(* IEC 61131-3 sources: TIA2AX/tests/V18/test_projects/expected/HW_2200330/ST10_PLC, 7 files *)

(* ---- HwIdentifiers.st ---- *)
TYPE
	HwIdentifiers : WORD
	(
		ST10_PLC_Rail_0 :=	WORD#256,
		ST10_PLC :=	WORD#48,
		ST10_PLC_Card_reader_writer_1 :=	WORD#51,
		ST10_PLC_CPU_display_1 :=	WORD#54,
		ST10_PLC_OPC_UA_1 :=	WORD#117,
		ST10_PLC_DP_interface_1 :=	WORD#60,
		ST10_PLC_PROFINET_interface_1 :=	WORD#64,
		ST10_PLC_PROFINET_interface_1_Port_1 :=	WORD#65,
		ST10_PLC_PROFINET_interface_1_Port_2 :=	WORD#66,
		ST10_PLC_PROFINET_interface_2 :=	WORD#72,
		ST10_PLC_PROFINET_interface_2_Port_1 :=	WORD#73,
		ST10_Switch_SCALANCE_X_rack :=	WORD#479,
		ST10_Switch :=	WORD#480,
		ST10_Switch_ST10_Switch :=	WORD#481,
		ST10_Switch_SCALANCE_interface_1 :=	WORD#482,
		ST10_Switch_SCALANCE_interface_1_Port_1 :=	WORD#483,
		ST10_Switch_SCALANCE_interface_1_Port_2 :=	WORD#484,
		ST10_Switch_SCALANCE_interface_1_Port_3 :=	WORD#485,
		ST10_Switch_SCALANCE_interface_1_Port_4 :=	WORD#486,
		ST10_Switch_SCALANCE_interface_1_Port_5 :=	WORD#487,
		ST10_Switch_SCALANCE_interface_1_Port_6 :=	WORD#488,
		ST10_Switch_SCALANCE_interface_1_Port_7 :=	WORD#489,
		ST10_Switch_SCALANCE_interface_1_Port_8 :=	WORD#490,
		ST10_Switch_SCALANCE_interface_1_Port_9 :=	WORD#491,
		ST10_Switch_SCALANCE_interface_1_Port_10 :=	WORD#492,
		ST10_Switch_SCALANCE_interface_1_Port_11 :=	WORD#493,
		ST10_Switch_SCALANCE_interface_1_Port_12 :=	WORD#494,
		ST10_Switch_SCALANCE_interface_1_Port_13 :=	WORD#495,
		ST10_Switch_SCALANCE_interface_1_Port_14 :=	WORD#496,
		ST10_Switch_SCALANCE_interface_1_Port_15 :=	WORD#497,
		ST10_Switch_SCALANCE_interface_1_Port_16 :=	WORD#498,
		ST10_ET200SP_Rack_0 :=	WORD#395,
		ST10_ET200SP :=	WORD#396,
		ST10_ET200SP_ST10_ET200SP :=	WORD#397,
		ST10_ET200SP_PROFINET_interface :=	WORD#259,
		ST10_ET200SP_PROFINET_interface_Port_1 :=	WORD#260,
		ST10_ET200SP_PROFINET_interface_Port_2 :=	WORD#261,
		ST10_ET200SP_BA_2xRJ45 :=	WORD#260,
		ST10_ET200SP_CM_AS_i_Master_ST_1 :=	WORD#274,
		ST10_ET200SP_DI_8x24VDC_ST_1 :=	WORD#264,
		ST10_ET200SP_DI_16x24VDC_ST_2 :=	WORD#265,
		ST10_ET200SP_DI_16x24VDC_ST_3 :=	WORD#266,
		ST10_ET200SP_DI_8x24VDC_ST_2 :=	WORD#267,
		ST10_ET200SP_DQ_8x24VDC_0_5A_ST_1 :=	WORD#268,
		ST10_ET200SP_DQ_8x24VDC_0_5A_ST_2 :=	WORD#269,
		ST10_ET200SP_DQ_8x24VDC_0_5A_ST_3 :=	WORD#270,
		ST10_ET200SP_DQ_8x24VDC_0_5A_ST_4 :=	WORD#271,
		ST10_ET200SP_CM_4xIO_Link_1 :=	WORD#272,
		ST10_ET200SP_Servermodul_1 :=	WORD#273,
		ST10_ET200SP_2_Rack_0 :=	WORD#399,
		ST10_ET200SP_2 :=	WORD#400,
		ST10_ET200SP_2_ST10_ET200SP_2 :=	WORD#401,
		ST10_ET200SP_2_PROFINET_interface :=	WORD#402,
		ST10_ET200SP_2_PROFINET_interface_Port_1 :=	WORD#404,
		ST10_ET200SP_2_PROFINET_interface_Port_2 :=	WORD#403,
		ST10_ET200SP_2_BA_2xRJ45 :=	WORD#404,
		ST10_ET200SP_2_21FM1 :=	WORD#405,
		ST10_ET200SP_2_21FM2 :=	WORD#406,
		ST10_ET200SP_2_21FM3 :=	WORD#407,
		ST10_ET200SP_2_21FM4 :=	WORD#408,
		ST10_ET200SP_2_21FM5 :=	WORD#409,
		ST10_ET200SP_2_21FM6 :=	WORD#410,
		ST10_ET200SP_2_21FM7 :=	WORD#411,
		ST10_ET200SP_2_21FM8 :=	WORD#412,
		ST10_ET200SP_2_21FM9 :=	WORD#413,
		ST10_ET200SP_2_21FM10 :=	WORD#414,
		ST10_ET200SP_2_21FM11 :=	WORD#415,
		ST10_ET200SP_2_21FM12 :=	WORD#416,
		ST10_ET200SP_2_22FM1 :=	WORD#417,
		ST10_ET200SP_2_22FM2 :=	WORD#418,
		ST10_ET200SP_2_22FM3 :=	WORD#419,
		ST10_ET200SP_2_22FM4 :=	WORD#420,
		ST10_ET200SP_2_22FM5 :=	WORD#421,
		ST10_ET200SP_2_22FM6 :=	WORD#422,
		ST10_ET200SP_2_22FM7 :=	WORD#423,
		ST10_ET200SP_2_22FM8 :=	WORD#424,
		ST10_ET200SP_2_22FM9 :=	WORD#425,
		ST10_ET200SP_2_22FM10 :=	WORD#426,
		ST10_ET200SP_2_22FM11 :=	WORD#427,
		ST10_ET200SP_2_22FM12 :=	WORD#428,
		ST10_ET200SP_2_22FM13 :=	WORD#429,
		ST10_ET200SP_2_Servermodul :=	WORD#430,
		ST10_CPX_PN_IO_Interface :=	WORD#434,
		ST10_CPX_PN_IO_Interface_Port_1 :=	WORD#435,
		ST10_CPX_PN_IO_Interface_Port_2 :=	WORD#436,
		ST10_CPX_CPX :=	WORD#437,
		ST10_CPX_MPA1S_VMPA1_FB_EMS_8_8DO_1 :=	WORD#438,
		ST10_CPX_MPA2G_VMPA2_FB_EMG_4_4DO_1 :=	WORD#439,
		ST10_1_DM260_Rack :=	WORD#441,
		ST10_1_DM260 :=	WORD#442,
		ST10_1_DM260_Interface :=	WORD#443,
		ST10_1_DM260_Interface_Port_1 :=	WORD#444,
		ST10_1_DM260_DataMan_260 :=	WORD#445,
		ST10_1_DM260_Acquisition_Control_1 :=	WORD#446,
		ST10_1_DM260_Acquisition_Status_1 :=	WORD#447,
		ST10_1_DM260_Results_Control_1 :=	WORD#448,
		ST10_1_DM260_Results_Status_1 :=	WORD#449,
		ST10_1_DM260_Soft_Event_Control_1 :=	WORD#450,
		ST10_1_DM260_User_Data_64_bytes_1 :=	WORD#451,
		ST10_1_DM260_Result_Data_64_bytes_1 :=	WORD#452,
		ST10_1_DM260_Turned_Rack :=	WORD#454,
		ST10_1_DM260_Turned :=	WORD#455,
		ST10_1_DM260_Turned_Interface :=	WORD#456,
		ST10_1_DM260_Turned_Interface_Port_1 :=	WORD#457,
		ST10_1_DM260_Turned_DataMan_260 :=	WORD#458,
		ST10_1_DM260_Turned_Acquisition_Control_1 :=	WORD#459,
		ST10_1_DM260_Turned_Acquisition_Status_1 :=	WORD#460,
		ST10_1_DM260_Turned_Results_Control_1 :=	WORD#461,
		ST10_1_DM260_Turned_Results_Status_1 :=	WORD#462,
		ST10_1_DM260_Turned_Soft_Event_Control_1 :=	WORD#463,
		ST10_1_DM260_Turned_User_Data_64_bytes_1 :=	WORD#464,
		ST10_1_DM260_Turned_Result_Data_64_bytes_1 :=	WORD#465,
		NONE:= WORD#0
	);
END_TYPE

(* ---- HwInputs.st ---- *)
TYPE
	HwInputs : STRUCT
		ST10_ET200SP_CM_AS_i_Master_ST_1 AT %B300 : ARRAY[0..63] OF BYTE;
		ST10_ET200SP_DI_8x24VDC_ST_1 AT %B0 : BYTE;
		ST10_ET200SP_DI_16x24VDC_ST_2 AT %B1 : WORD;
		ST10_ET200SP_DI_16x24VDC_ST_3 AT %B3 : WORD;
		ST10_ET200SP_DI_8x24VDC_ST_2 AT %B5 : BYTE;
		ST10_ET200SP_CM_4xIO_Link_1 AT %B100 : ARRAY[0..31] OF BYTE;
		ST10_ET200SP_2_21FM1 AT %B600 : DWORD;
		ST10_ET200SP_2_21FM2 AT %B604 : DWORD;
		ST10_ET200SP_2_21FM3 AT %B652 : DWORD;
		ST10_ET200SP_2_21FM4 AT %B612 : DWORD;
		ST10_ET200SP_2_21FM5 AT %B616 : DWORD;
		ST10_ET200SP_2_21FM6 AT %B620 : DWORD;
		ST10_ET200SP_2_21FM7 AT %B624 : DWORD;
		ST10_ET200SP_2_21FM8 AT %B628 : DWORD;
		ST10_ET200SP_2_21FM9 AT %B632 : DWORD;
		ST10_ET200SP_2_21FM10 AT %B636 : DWORD;
		ST10_ET200SP_2_21FM11 AT %B640 : DWORD;
		ST10_ET200SP_2_21FM12 AT %B644 : DWORD;
		ST10_ET200SP_2_22FM1 AT %B648 : DWORD;
		ST10_ET200SP_2_22FM2 AT %B608 : DWORD;
		ST10_ET200SP_2_22FM3 AT %B696 : DWORD;
		ST10_ET200SP_2_22FM4 AT %B660 : DWORD;
		ST10_ET200SP_2_22FM5 AT %B664 : DWORD;
		ST10_ET200SP_2_22FM6 AT %B668 : DWORD;
		ST10_ET200SP_2_22FM7 AT %B672 : DWORD;
		ST10_ET200SP_2_22FM8 AT %B676 : DWORD;
		ST10_ET200SP_2_22FM9 AT %B656 : DWORD;
		ST10_ET200SP_2_22FM10 AT %B684 : DWORD;
		ST10_ET200SP_2_22FM11 AT %B688 : DWORD;
		ST10_ET200SP_2_22FM12 AT %B692 : DWORD;
		ST10_ET200SP_2_22FM13 AT %B680 : DWORD;
		ST10_1_DM260_Acquisition_Status_1 AT %B1000 : ARRAY[0..2] OF BYTE;
		ST10_1_DM260_Results_Status_1 AT %B1003 : BYTE;
		ST10_1_DM260_Soft_Event_Control_1 AT %B1004 : BYTE;
		ST10_1_DM260_Result_Data_64_bytes_1 AT %B1010 : ARRAY[0..71] OF BYTE;
		ST10_1_DM260_Turned_Acquisition_Status_1 AT %B1200 : ARRAY[0..2] OF BYTE;
		ST10_1_DM260_Turned_Results_Status_1 AT %B1203 : BYTE;
		ST10_1_DM260_Turned_Soft_Event_Control_1 AT %B1204 : BYTE;
		ST10_1_DM260_Turned_Result_Data_64_bytes_1 AT %B1210 : ARRAY[0..71] OF BYTE;
	END_STRUCT;
END_TYPE

(* ---- HwOutputs.st ---- *)
TYPE
	HwOutputs : STRUCT
		ST10_ET200SP_CM_AS_i_Master_ST_1 AT %B300 : ARRAY[0..63] OF BYTE;
		ST10_ET200SP_DQ_8x24VDC_0_5A_ST_1 AT %B0 : BYTE;
		ST10_ET200SP_DQ_8x24VDC_0_5A_ST_2 AT %B1 : BYTE;
		ST10_ET200SP_DQ_8x24VDC_0_5A_ST_3 AT %B2 : BYTE;
		ST10_ET200SP_DQ_8x24VDC_0_5A_ST_4 AT %B3 : BYTE;
		ST10_ET200SP_CM_4xIO_Link_1 AT %B100 : ARRAY[0..31] OF BYTE;
		ST10_ET200SP_2_21FM1 AT %B600 : WORD;
		ST10_ET200SP_2_21FM2 AT %B604 : WORD;
		ST10_ET200SP_2_21FM3 AT %B652 : WORD;
		ST10_ET200SP_2_21FM4 AT %B612 : WORD;
		ST10_ET200SP_2_21FM5 AT %B616 : WORD;
		ST10_ET200SP_2_21FM6 AT %B620 : WORD;
		ST10_ET200SP_2_21FM7 AT %B624 : WORD;
		ST10_ET200SP_2_21FM8 AT %B628 : WORD;
		ST10_ET200SP_2_21FM9 AT %B632 : WORD;
		ST10_ET200SP_2_21FM10 AT %B636 : WORD;
		ST10_ET200SP_2_21FM11 AT %B640 : WORD;
		ST10_ET200SP_2_21FM12 AT %B644 : WORD;
		ST10_ET200SP_2_22FM1 AT %B648 : WORD;
		ST10_ET200SP_2_22FM2 AT %B608 : WORD;
		ST10_ET200SP_2_22FM3 AT %B692 : WORD;
		ST10_ET200SP_2_22FM4 AT %B660 : WORD;
		ST10_ET200SP_2_22FM5 AT %B664 : WORD;
		ST10_ET200SP_2_22FM6 AT %B668 : WORD;
		ST10_ET200SP_2_22FM7 AT %B672 : WORD;
		ST10_ET200SP_2_22FM8 AT %B676 : WORD;
		ST10_ET200SP_2_22FM9 AT %B656 : WORD;
		ST10_ET200SP_2_22FM10 AT %B684 : WORD;
		ST10_ET200SP_2_22FM11 AT %B688 : WORD;
		ST10_ET200SP_2_22FM12 AT %B690 : WORD;
		ST10_ET200SP_2_22FM13 AT %B680 : WORD;
		ST10_CPX_MPA1S_VMPA1_FB_EMS_8_8DO_1 AT %B200 : BYTE;
		ST10_CPX_MPA2G_VMPA2_FB_EMG_4_4DO_1 AT %B201 : BYTE;
		ST10_1_DM260_Acquisition_Control_1 AT %B1000 : BYTE;
		ST10_1_DM260_Results_Control_1 AT %B1001 : BYTE;
		ST10_1_DM260_Soft_Event_Control_1 AT %B1002 : BYTE;
		ST10_1_DM260_User_Data_64_bytes_1 AT %B1010 : ARRAY[0..67] OF BYTE;
		ST10_1_DM260_Turned_Acquisition_Control_1 AT %B1200 : BYTE;
		ST10_1_DM260_Turned_Results_Control_1 AT %B1203 : BYTE;
		ST10_1_DM260_Turned_Soft_Event_Control_1 AT %B1204 : BYTE;
		ST10_1_DM260_Turned_User_Data_64_bytes_1 AT %B1210 : ARRAY[0..67] OF BYTE;
	END_STRUCT;
END_TYPE

(* ---- PlcInputs.st ---- *)
TYPE
	PlcInputs : STRUCT
		ST10_ET200SP_CM_AS_i_Master_ST_1 : ARRAY[0..63] OF BYTE;
		ST10_ET200SP_DI_8x24VDC_ST_1 : BYTE;
		ST10_ET200SP_DI_16x24VDC_ST_2 : WORD;
		ST10_ET200SP_DI_16x24VDC_ST_3 : WORD;
		ST10_ET200SP_DI_8x24VDC_ST_2 : BYTE;
		ST10_ET200SP_CM_4xIO_Link_1 : ARRAY[0..31] OF BYTE;
		ST10_ET200SP_2_21FM1 : DWORD;
		ST10_ET200SP_2_21FM2 : DWORD;
		ST10_ET200SP_2_21FM3 : DWORD;
		ST10_ET200SP_2_21FM4 : DWORD;
		ST10_ET200SP_2_21FM5 : DWORD;
		ST10_ET200SP_2_21FM6 : DWORD;
		ST10_ET200SP_2_21FM7 : DWORD;
		ST10_ET200SP_2_21FM8 : DWORD;
		ST10_ET200SP_2_21FM9 : DWORD;
		ST10_ET200SP_2_21FM10 : DWORD;
		ST10_ET200SP_2_21FM11 : DWORD;
		ST10_ET200SP_2_21FM12 : DWORD;
		ST10_ET200SP_2_22FM1 : DWORD;
		ST10_ET200SP_2_22FM2 : DWORD;
		ST10_ET200SP_2_22FM3 : DWORD;
		ST10_ET200SP_2_22FM4 : DWORD;
		ST10_ET200SP_2_22FM5 : DWORD;
		ST10_ET200SP_2_22FM6 : DWORD;
		ST10_ET200SP_2_22FM7 : DWORD;
		ST10_ET200SP_2_22FM8 : DWORD;
		ST10_ET200SP_2_22FM9 : DWORD;
		ST10_ET200SP_2_22FM10 : DWORD;
		ST10_ET200SP_2_22FM11 : DWORD;
		ST10_ET200SP_2_22FM12 : DWORD;
		ST10_ET200SP_2_22FM13 : DWORD;
		ST10_1_DM260_Acquisition_Status_1 : ARRAY[0..2] OF BYTE;
		ST10_1_DM260_Results_Status_1 : BYTE;
		ST10_1_DM260_Soft_Event_Control_1 : BYTE;
		ST10_1_DM260_Result_Data_64_bytes_1 : ARRAY[0..71] OF BYTE;
		ST10_1_DM260_Turned_Acquisition_Status_1 : ARRAY[0..2] OF BYTE;
		ST10_1_DM260_Turned_Results_Status_1 : BYTE;
		ST10_1_DM260_Turned_Soft_Event_Control_1 : BYTE;
		ST10_1_DM260_Turned_Result_Data_64_bytes_1 : ARRAY[0..71] OF BYTE;
	END_STRUCT;
END_TYPE

(* ---- PlcOutputs.st ---- *)
TYPE
	PlcOutputs : STRUCT
		ST10_ET200SP_CM_AS_i_Master_ST_1 : ARRAY[0..63] OF BYTE;
		ST10_ET200SP_DQ_8x24VDC_0_5A_ST_1 : BYTE;
		ST10_ET200SP_DQ_8x24VDC_0_5A_ST_2 : BYTE;
		ST10_ET200SP_DQ_8x24VDC_0_5A_ST_3 : BYTE;
		ST10_ET200SP_DQ_8x24VDC_0_5A_ST_4 : BYTE;
		ST10_ET200SP_CM_4xIO_Link_1 : ARRAY[0..31] OF BYTE;
		ST10_ET200SP_2_21FM1 : WORD;
		ST10_ET200SP_2_21FM2 : WORD;
		ST10_ET200SP_2_21FM3 : WORD;
		ST10_ET200SP_2_21FM4 : WORD;
		ST10_ET200SP_2_21FM5 : WORD;
		ST10_ET200SP_2_21FM6 : WORD;
		ST10_ET200SP_2_21FM7 : WORD;
		ST10_ET200SP_2_21FM8 : WORD;
		ST10_ET200SP_2_21FM9 : WORD;
		ST10_ET200SP_2_21FM10 : WORD;
		ST10_ET200SP_2_21FM11 : WORD;
		ST10_ET200SP_2_21FM12 : WORD;
		ST10_ET200SP_2_22FM1 : WORD;
		ST10_ET200SP_2_22FM2 : WORD;
		ST10_ET200SP_2_22FM3 : WORD;
		ST10_ET200SP_2_22FM4 : WORD;
		ST10_ET200SP_2_22FM5 : WORD;
		ST10_ET200SP_2_22FM6 : WORD;
		ST10_ET200SP_2_22FM7 : WORD;
		ST10_ET200SP_2_22FM8 : WORD;
		ST10_ET200SP_2_22FM9 : WORD;
		ST10_ET200SP_2_22FM10 : WORD;
		ST10_ET200SP_2_22FM11 : WORD;
		ST10_ET200SP_2_22FM12 : WORD;
		ST10_ET200SP_2_22FM13 : WORD;
		ST10_CPX_MPA1S_VMPA1_FB_EMS_8_8DO_1 : BYTE;
		ST10_CPX_MPA2G_VMPA2_FB_EMG_4_4DO_1 : BYTE;
		ST10_1_DM260_Acquisition_Control_1 : BYTE;
		ST10_1_DM260_Results_Control_1 : BYTE;
		ST10_1_DM260_Soft_Event_Control_1 : BYTE;
		ST10_1_DM260_User_Data_64_bytes_1 : ARRAY[0..67] OF BYTE;
		ST10_1_DM260_Turned_Acquisition_Control_1 : BYTE;
		ST10_1_DM260_Turned_Results_Control_1 : BYTE;
		ST10_1_DM260_Turned_Soft_Event_Control_1 : BYTE;
		ST10_1_DM260_Turned_User_Data_64_bytes_1 : ARRAY[0..67] OF BYTE;
	END_STRUCT;
END_TYPE

(* ---- CopyInputs.st ---- *)
FUNCTION CopyInputs
	VAR_EXTERNAL
		HwInputs : HwInputs;
		PlcInputs : PlcInputs;
	END_VAR
	PlcInputs.ST10_ET200SP_CM_AS_i_Master_ST_1[0] := HwInputs.ST10_ET200SP_CM_AS_i_Master_ST_1[0];
	PlcInputs.ST10_ET200SP_CM_AS_i_Master_ST_1[1] := HwInputs.ST10_ET200SP_CM_AS_i_Master_ST_1[1];
	PlcInputs.ST10_ET200SP_CM_AS_i_Master_ST_1[2] := HwInputs.ST10_ET200SP_CM_AS_i_Master_ST_1[2];
	PlcInputs.ST10_ET200SP_CM_AS_i_Master_ST_1[3] := HwInputs.ST10_ET200SP_CM_AS_i_Master_ST_1[3];
	PlcInputs.ST10_ET200SP_CM_AS_i_Master_ST_1[4] := HwInputs.ST10_ET200SP_CM_AS_i_Master_ST_1[4];
	PlcInputs.ST10_ET200SP_CM_AS_i_Master_ST_1[5] := HwInputs.ST10_ET200SP_CM_AS_i_Master_ST_1[5];
	PlcInputs.ST10_ET200SP_CM_AS_i_Master_ST_1[6] := HwInputs.ST10_ET200SP_CM_AS_i_Master_ST_1[6];
	PlcInputs.ST10_ET200SP_CM_AS_i_Master_ST_1[7] := HwInputs.ST10_ET200SP_CM_AS_i_Master_ST_1[7];
	PlcInputs.ST10_ET200SP_CM_AS_i_Master_ST_1[8] := HwInputs.ST10_ET200SP_CM_AS_i_Master_ST_1[8];
	PlcInputs.ST10_ET200SP_CM_AS_i_Master_ST_1[9] := HwInputs.ST10_ET200SP_CM_AS_i_Master_ST_1[9];
	PlcInputs.ST10_ET200SP_CM_AS_i_Master_ST_1[10] := HwInputs.ST10_ET200SP_CM_AS_i_Master_ST_1[10];
	PlcInputs.ST10_ET200SP_CM_AS_i_Master_ST_1[11] := HwInputs.ST10_ET200SP_CM_AS_i_Master_ST_1[11];
	PlcInputs.ST10_ET200SP_CM_AS_i_Master_ST_1[12] := HwInputs.ST10_ET200SP_CM_AS_i_Master_ST_1[12];
	PlcInputs.ST10_ET200SP_CM_AS_i_Master_ST_1[13] := HwInputs.ST10_ET200SP_CM_AS_i_Master_ST_1[13];
	PlcInputs.ST10_ET200SP_CM_AS_i_Master_ST_1[14] := HwInputs.ST10_ET200SP_CM_AS_i_Master_ST_1[14];
	PlcInputs.ST10_ET200SP_CM_AS_i_Master_ST_1[15] := HwInputs.ST10_ET200SP_CM_AS_i_Master_ST_1[15];
	PlcInputs.ST10_ET200SP_CM_AS_i_Master_ST_1[16] := HwInputs.ST10_ET200SP_CM_AS_i_Master_ST_1[16];
	PlcInputs.ST10_ET200SP_CM_AS_i_Master_ST_1[17] := HwInputs.ST10_ET200SP_CM_AS_i_Master_ST_1[17];
	PlcInputs.ST10_ET200SP_CM_AS_i_Master_ST_1[18] := HwInputs.ST10_ET200SP_CM_AS_i_Master_ST_1[18];
	PlcInputs.ST10_ET200SP_CM_AS_i_Master_ST_1[19] := HwInputs.ST10_ET200SP_CM_AS_i_Master_ST_1[19];
	PlcInputs.ST10_ET200SP_CM_AS_i_Master_ST_1[20] := HwInputs.ST10_ET200SP_CM_AS_i_Master_ST_1[20];
	PlcInputs.ST10_ET200SP_CM_AS_i_Master_ST_1[21] := HwInputs.ST10_ET200SP_CM_AS_i_Master_ST_1[21];
	PlcInputs.ST10_ET200SP_CM_AS_i_Master_ST_1[22] := HwInputs.ST10_ET200SP_CM_AS_i_Master_ST_1[22];
	PlcInputs.ST10_ET200SP_CM_AS_i_Master_ST_1[23] := HwInputs.ST10_ET200SP_CM_AS_i_Master_ST_1[23];
	PlcInputs.ST10_ET200SP_CM_AS_i_Master_ST_1[24] := HwInputs.ST10_ET200SP_CM_AS_i_Master_ST_1[24];
	PlcInputs.ST10_ET200SP_CM_AS_i_Master_ST_1[25] := HwInputs.ST10_ET200SP_CM_AS_i_Master_ST_1[25];
	PlcInputs.ST10_ET200SP_CM_AS_i_Master_ST_1[26] := HwInputs.ST10_ET200SP_CM_AS_i_Master_ST_1[26];
	PlcInputs.ST10_ET200SP_CM_AS_i_Master_ST_1[27] := HwInputs.ST10_ET200SP_CM_AS_i_Master_ST_1[27];
	PlcInputs.ST10_ET200SP_CM_AS_i_Master_ST_1[28] := HwInputs.ST10_ET200SP_CM_AS_i_Master_ST_1[28];
	PlcInputs.ST10_ET200SP_CM_AS_i_Master_ST_1[29] := HwInputs.ST10_ET200SP_CM_AS_i_Master_ST_1[29];
	PlcInputs.ST10_ET200SP_CM_AS_i_Master_ST_1[30] := HwInputs.ST10_ET200SP_CM_AS_i_Master_ST_1[30];
	PlcInputs.ST10_ET200SP_CM_AS_i_Master_ST_1[31] := HwInputs.ST10_ET200SP_CM_AS_i_Master_ST_1[31];
	PlcInputs.ST10_ET200SP_CM_AS_i_Master_ST_1[32] := HwInputs.ST10_ET200SP_CM_AS_i_Master_ST_1[32];
	PlcInputs.ST10_ET200SP_CM_AS_i_Master_ST_1[33] := HwInputs.ST10_ET200SP_CM_AS_i_Master_ST_1[33];
	PlcInputs.ST10_ET200SP_CM_AS_i_Master_ST_1[34] := HwInputs.ST10_ET200SP_CM_AS_i_Master_ST_1[34];
	PlcInputs.ST10_ET200SP_CM_AS_i_Master_ST_1[35] := HwInputs.ST10_ET200SP_CM_AS_i_Master_ST_1[35];
	PlcInputs.ST10_ET200SP_CM_AS_i_Master_ST_1[36] := HwInputs.ST10_ET200SP_CM_AS_i_Master_ST_1[36];
	PlcInputs.ST10_ET200SP_CM_AS_i_Master_ST_1[37] := HwInputs.ST10_ET200SP_CM_AS_i_Master_ST_1[37];
	PlcInputs.ST10_ET200SP_CM_AS_i_Master_ST_1[38] := HwInputs.ST10_ET200SP_CM_AS_i_Master_ST_1[38];
	PlcInputs.ST10_ET200SP_CM_AS_i_Master_ST_1[39] := HwInputs.ST10_ET200SP_CM_AS_i_Master_ST_1[39];
	PlcInputs.ST10_ET200SP_CM_AS_i_Master_ST_1[40] := HwInputs.ST10_ET200SP_CM_AS_i_Master_ST_1[40];
	PlcInputs.ST10_ET200SP_CM_AS_i_Master_ST_1[41] := HwInputs.ST10_ET200SP_CM_AS_i_Master_ST_1[41];
	PlcInputs.ST10_ET200SP_CM_AS_i_Master_ST_1[42] := HwInputs.ST10_ET200SP_CM_AS_i_Master_ST_1[42];
	PlcInputs.ST10_ET200SP_CM_AS_i_Master_ST_1[43] := HwInputs.ST10_ET200SP_CM_AS_i_Master_ST_1[43];
	PlcInputs.ST10_ET200SP_CM_AS_i_Master_ST_1[44] := HwInputs.ST10_ET200SP_CM_AS_i_Master_ST_1[44];
	PlcInputs.ST10_ET200SP_CM_AS_i_Master_ST_1[45] := HwInputs.ST10_ET200SP_CM_AS_i_Master_ST_1[45];
	PlcInputs.ST10_ET200SP_CM_AS_i_Master_ST_1[46] := HwInputs.ST10_ET200SP_CM_AS_i_Master_ST_1[46];
	PlcInputs.ST10_ET200SP_CM_AS_i_Master_ST_1[47] := HwInputs.ST10_ET200SP_CM_AS_i_Master_ST_1[47];
	PlcInputs.ST10_ET200SP_CM_AS_i_Master_ST_1[48] := HwInputs.ST10_ET200SP_CM_AS_i_Master_ST_1[48];
	PlcInputs.ST10_ET200SP_CM_AS_i_Master_ST_1[49] := HwInputs.ST10_ET200SP_CM_AS_i_Master_ST_1[49];
	PlcInputs.ST10_ET200SP_CM_AS_i_Master_ST_1[50] := HwInputs.ST10_ET200SP_CM_AS_i_Master_ST_1[50];
	PlcInputs.ST10_ET200SP_CM_AS_i_Master_ST_1[51] := HwInputs.ST10_ET200SP_CM_AS_i_Master_ST_1[51];
	PlcInputs.ST10_ET200SP_CM_AS_i_Master_ST_1[52] := HwInputs.ST10_ET200SP_CM_AS_i_Master_ST_1[52];
	PlcInputs.ST10_ET200SP_CM_AS_i_Master_ST_1[53] := HwInputs.ST10_ET200SP_CM_AS_i_Master_ST_1[53];
	PlcInputs.ST10_ET200SP_CM_AS_i_Master_ST_1[54] := HwInputs.ST10_ET200SP_CM_AS_i_Master_ST_1[54];
	PlcInputs.ST10_ET200SP_CM_AS_i_Master_ST_1[55] := HwInputs.ST10_ET200SP_CM_AS_i_Master_ST_1[55];
	PlcInputs.ST10_ET200SP_CM_AS_i_Master_ST_1[56] := HwInputs.ST10_ET200SP_CM_AS_i_Master_ST_1[56];
	PlcInputs.ST10_ET200SP_CM_AS_i_Master_ST_1[57] := HwInputs.ST10_ET200SP_CM_AS_i_Master_ST_1[57];
	PlcInputs.ST10_ET200SP_CM_AS_i_Master_ST_1[58] := HwInputs.ST10_ET200SP_CM_AS_i_Master_ST_1[58];
	PlcInputs.ST10_ET200SP_CM_AS_i_Master_ST_1[59] := HwInputs.ST10_ET200SP_CM_AS_i_Master_ST_1[59];
	PlcInputs.ST10_ET200SP_CM_AS_i_Master_ST_1[60] := HwInputs.ST10_ET200SP_CM_AS_i_Master_ST_1[60];
	PlcInputs.ST10_ET200SP_CM_AS_i_Master_ST_1[61] := HwInputs.ST10_ET200SP_CM_AS_i_Master_ST_1[61];
	PlcInputs.ST10_ET200SP_CM_AS_i_Master_ST_1[62] := HwInputs.ST10_ET200SP_CM_AS_i_Master_ST_1[62];
	PlcInputs.ST10_ET200SP_CM_AS_i_Master_ST_1[63] := HwInputs.ST10_ET200SP_CM_AS_i_Master_ST_1[63];
	PlcInputs.ST10_ET200SP_DI_8x24VDC_ST_1 := HwInputs.ST10_ET200SP_DI_8x24VDC_ST_1;
	PlcInputs.ST10_ET200SP_DI_16x24VDC_ST_2 := HwInputs.ST10_ET200SP_DI_16x24VDC_ST_2;
	PlcInputs.ST10_ET200SP_DI_16x24VDC_ST_3 := HwInputs.ST10_ET200SP_DI_16x24VDC_ST_3;
	PlcInputs.ST10_ET200SP_DI_8x24VDC_ST_2 := HwInputs.ST10_ET200SP_DI_8x24VDC_ST_2;
	PlcInputs.ST10_ET200SP_CM_4xIO_Link_1[0] := HwInputs.ST10_ET200SP_CM_4xIO_Link_1[0];
	PlcInputs.ST10_ET200SP_CM_4xIO_Link_1[1] := HwInputs.ST10_ET200SP_CM_4xIO_Link_1[1];
	PlcInputs.ST10_ET200SP_CM_4xIO_Link_1[2] := HwInputs.ST10_ET200SP_CM_4xIO_Link_1[2];
	PlcInputs.ST10_ET200SP_CM_4xIO_Link_1[3] := HwInputs.ST10_ET200SP_CM_4xIO_Link_1[3];
	PlcInputs.ST10_ET200SP_CM_4xIO_Link_1[4] := HwInputs.ST10_ET200SP_CM_4xIO_Link_1[4];
	PlcInputs.ST10_ET200SP_CM_4xIO_Link_1[5] := HwInputs.ST10_ET200SP_CM_4xIO_Link_1[5];
	PlcInputs.ST10_ET200SP_CM_4xIO_Link_1[6] := HwInputs.ST10_ET200SP_CM_4xIO_Link_1[6];
	PlcInputs.ST10_ET200SP_CM_4xIO_Link_1[7] := HwInputs.ST10_ET200SP_CM_4xIO_Link_1[7];
	PlcInputs.ST10_ET200SP_CM_4xIO_Link_1[8] := HwInputs.ST10_ET200SP_CM_4xIO_Link_1[8];
	PlcInputs.ST10_ET200SP_CM_4xIO_Link_1[9] := HwInputs.ST10_ET200SP_CM_4xIO_Link_1[9];
	PlcInputs.ST10_ET200SP_CM_4xIO_Link_1[10] := HwInputs.ST10_ET200SP_CM_4xIO_Link_1[10];
	PlcInputs.ST10_ET200SP_CM_4xIO_Link_1[11] := HwInputs.ST10_ET200SP_CM_4xIO_Link_1[11];
	PlcInputs.ST10_ET200SP_CM_4xIO_Link_1[12] := HwInputs.ST10_ET200SP_CM_4xIO_Link_1[12];
	PlcInputs.ST10_ET200SP_CM_4xIO_Link_1[13] := HwInputs.ST10_ET200SP_CM_4xIO_Link_1[13];
	PlcInputs.ST10_ET200SP_CM_4xIO_Link_1[14] := HwInputs.ST10_ET200SP_CM_4xIO_Link_1[14];
	PlcInputs.ST10_ET200SP_CM_4xIO_Link_1[15] := HwInputs.ST10_ET200SP_CM_4xIO_Link_1[15];
	PlcInputs.ST10_ET200SP_CM_4xIO_Link_1[16] := HwInputs.ST10_ET200SP_CM_4xIO_Link_1[16];
	PlcInputs.ST10_ET200SP_CM_4xIO_Link_1[17] := HwInputs.ST10_ET200SP_CM_4xIO_Link_1[17];
	PlcInputs.ST10_ET200SP_CM_4xIO_Link_1[18] := HwInputs.ST10_ET200SP_CM_4xIO_Link_1[18];
	PlcInputs.ST10_ET200SP_CM_4xIO_Link_1[19] := HwInputs.ST10_ET200SP_CM_4xIO_Link_1[19];
	PlcInputs.ST10_ET200SP_CM_4xIO_Link_1[20] := HwInputs.ST10_ET200SP_CM_4xIO_Link_1[20];
	PlcInputs.ST10_ET200SP_CM_4xIO_Link_1[21] := HwInputs.ST10_ET200SP_CM_4xIO_Link_1[21];
	PlcInputs.ST10_ET200SP_CM_4xIO_Link_1[22] := HwInputs.ST10_ET200SP_CM_4xIO_Link_1[22];
	PlcInputs.ST10_ET200SP_CM_4xIO_Link_1[23] := HwInputs.ST10_ET200SP_CM_4xIO_Link_1[23];
	PlcInputs.ST10_ET200SP_CM_4xIO_Link_1[24] := HwInputs.ST10_ET200SP_CM_4xIO_Link_1[24];
	PlcInputs.ST10_ET200SP_CM_4xIO_Link_1[25] := HwInputs.ST10_ET200SP_CM_4xIO_Link_1[25];
	PlcInputs.ST10_ET200SP_CM_4xIO_Link_1[26] := HwInputs.ST10_ET200SP_CM_4xIO_Link_1[26];
	PlcInputs.ST10_ET200SP_CM_4xIO_Link_1[27] := HwInputs.ST10_ET200SP_CM_4xIO_Link_1[27];
	PlcInputs.ST10_ET200SP_CM_4xIO_Link_1[28] := HwInputs.ST10_ET200SP_CM_4xIO_Link_1[28];
	PlcInputs.ST10_ET200SP_CM_4xIO_Link_1[29] := HwInputs.ST10_ET200SP_CM_4xIO_Link_1[29];
	PlcInputs.ST10_ET200SP_CM_4xIO_Link_1[30] := HwInputs.ST10_ET200SP_CM_4xIO_Link_1[30];
	PlcInputs.ST10_ET200SP_CM_4xIO_Link_1[31] := HwInputs.ST10_ET200SP_CM_4xIO_Link_1[31];
	PlcInputs.ST10_ET200SP_2_21FM1 := HwInputs.ST10_ET200SP_2_21FM1;
	PlcInputs.ST10_ET200SP_2_21FM2 := HwInputs.ST10_ET200SP_2_21FM2;
	PlcInputs.ST10_ET200SP_2_21FM3 := HwInputs.ST10_ET200SP_2_21FM3;
	PlcInputs.ST10_ET200SP_2_21FM4 := HwInputs.ST10_ET200SP_2_21FM4;
	PlcInputs.ST10_ET200SP_2_21FM5 := HwInputs.ST10_ET200SP_2_21FM5;
	PlcInputs.ST10_ET200SP_2_21FM6 := HwInputs.ST10_ET200SP_2_21FM6;
	PlcInputs.ST10_ET200SP_2_21FM7 := HwInputs.ST10_ET200SP_2_21FM7;
	PlcInputs.ST10_ET200SP_2_21FM8 := HwInputs.ST10_ET200SP_2_21FM8;
	PlcInputs.ST10_ET200SP_2_21FM9 := HwInputs.ST10_ET200SP_2_21FM9;
	PlcInputs.ST10_ET200SP_2_21FM10 := HwInputs.ST10_ET200SP_2_21FM10;
	PlcInputs.ST10_ET200SP_2_21FM11 := HwInputs.ST10_ET200SP_2_21FM11;
	PlcInputs.ST10_ET200SP_2_21FM12 := HwInputs.ST10_ET200SP_2_21FM12;
	PlcInputs.ST10_ET200SP_2_22FM1 := HwInputs.ST10_ET200SP_2_22FM1;
	PlcInputs.ST10_ET200SP_2_22FM2 := HwInputs.ST10_ET200SP_2_22FM2;
	PlcInputs.ST10_ET200SP_2_22FM3 := HwInputs.ST10_ET200SP_2_22FM3;
	PlcInputs.ST10_ET200SP_2_22FM4 := HwInputs.ST10_ET200SP_2_22FM4;
	PlcInputs.ST10_ET200SP_2_22FM5 := HwInputs.ST10_ET200SP_2_22FM5;
	PlcInputs.ST10_ET200SP_2_22FM6 := HwInputs.ST10_ET200SP_2_22FM6;
	PlcInputs.ST10_ET200SP_2_22FM7 := HwInputs.ST10_ET200SP_2_22FM7;
	PlcInputs.ST10_ET200SP_2_22FM8 := HwInputs.ST10_ET200SP_2_22FM8;
	PlcInputs.ST10_ET200SP_2_22FM9 := HwInputs.ST10_ET200SP_2_22FM9;
	PlcInputs.ST10_ET200SP_2_22FM10 := HwInputs.ST10_ET200SP_2_22FM10;
	PlcInputs.ST10_ET200SP_2_22FM11 := HwInputs.ST10_ET200SP_2_22FM11;
	PlcInputs.ST10_ET200SP_2_22FM12 := HwInputs.ST10_ET200SP_2_22FM12;
	PlcInputs.ST10_ET200SP_2_22FM13 := HwInputs.ST10_ET200SP_2_22FM13;
	PlcInputs.ST10_1_DM260_Acquisition_Status_1[0] := HwInputs.ST10_1_DM260_Acquisition_Status_1[0];
	PlcInputs.ST10_1_DM260_Acquisition_Status_1[1] := HwInputs.ST10_1_DM260_Acquisition_Status_1[1];
	PlcInputs.ST10_1_DM260_Acquisition_Status_1[2] := HwInputs.ST10_1_DM260_Acquisition_Status_1[2];
	PlcInputs.ST10_1_DM260_Results_Status_1 := HwInputs.ST10_1_DM260_Results_Status_1;
	PlcInputs.ST10_1_DM260_Soft_Event_Control_1 := HwInputs.ST10_1_DM260_Soft_Event_Control_1;
	PlcInputs.ST10_1_DM260_Result_Data_64_bytes_1[0] := HwInputs.ST10_1_DM260_Result_Data_64_bytes_1[0];
	PlcInputs.ST10_1_DM260_Result_Data_64_bytes_1[1] := HwInputs.ST10_1_DM260_Result_Data_64_bytes_1[1];
	PlcInputs.ST10_1_DM260_Result_Data_64_bytes_1[2] := HwInputs.ST10_1_DM260_Result_Data_64_bytes_1[2];
	PlcInputs.ST10_1_DM260_Result_Data_64_bytes_1[3] := HwInputs.ST10_1_DM260_Result_Data_64_bytes_1[3];
	PlcInputs.ST10_1_DM260_Result_Data_64_bytes_1[4] := HwInputs.ST10_1_DM260_Result_Data_64_bytes_1[4];
	PlcInputs.ST10_1_DM260_Result_Data_64_bytes_1[5] := HwInputs.ST10_1_DM260_Result_Data_64_bytes_1[5];
	PlcInputs.ST10_1_DM260_Result_Data_64_bytes_1[6] := HwInputs.ST10_1_DM260_Result_Data_64_bytes_1[6];
	PlcInputs.ST10_1_DM260_Result_Data_64_bytes_1[7] := HwInputs.ST10_1_DM260_Result_Data_64_bytes_1[7];
	PlcInputs.ST10_1_DM260_Result_Data_64_bytes_1[8] := HwInputs.ST10_1_DM260_Result_Data_64_bytes_1[8];
	PlcInputs.ST10_1_DM260_Result_Data_64_bytes_1[9] := HwInputs.ST10_1_DM260_Result_Data_64_bytes_1[9];
	PlcInputs.ST10_1_DM260_Result_Data_64_bytes_1[10] := HwInputs.ST10_1_DM260_Result_Data_64_bytes_1[10];
	PlcInputs.ST10_1_DM260_Result_Data_64_bytes_1[11] := HwInputs.ST10_1_DM260_Result_Data_64_bytes_1[11];
	PlcInputs.ST10_1_DM260_Result_Data_64_bytes_1[12] := HwInputs.ST10_1_DM260_Result_Data_64_bytes_1[12];
	PlcInputs.ST10_1_DM260_Result_Data_64_bytes_1[13] := HwInputs.ST10_1_DM260_Result_Data_64_bytes_1[13];
	PlcInputs.ST10_1_DM260_Result_Data_64_bytes_1[14] := HwInputs.ST10_1_DM260_Result_Data_64_bytes_1[14];
	PlcInputs.ST10_1_DM260_Result_Data_64_bytes_1[15] := HwInputs.ST10_1_DM260_Result_Data_64_bytes_1[15];
	PlcInputs.ST10_1_DM260_Result_Data_64_bytes_1[16] := HwInputs.ST10_1_DM260_Result_Data_64_bytes_1[16];
	PlcInputs.ST10_1_DM260_Result_Data_64_bytes_1[17] := HwInputs.ST10_1_DM260_Result_Data_64_bytes_1[17];
	PlcInputs.ST10_1_DM260_Result_Data_64_bytes_1[18] := HwInputs.ST10_1_DM260_Result_Data_64_bytes_1[18];
	PlcInputs.ST10_1_DM260_Result_Data_64_bytes_1[19] := HwInputs.ST10_1_DM260_Result_Data_64_bytes_1[19];
	PlcInputs.ST10_1_DM260_Result_Data_64_bytes_1[20] := HwInputs.ST10_1_DM260_Result_Data_64_bytes_1[20];
	PlcInputs.ST10_1_DM260_Result_Data_64_bytes_1[21] := HwInputs.ST10_1_DM260_Result_Data_64_bytes_1[21];
	PlcInputs.ST10_1_DM260_Result_Data_64_bytes_1[22] := HwInputs.ST10_1_DM260_Result_Data_64_bytes_1[22];
	PlcInputs.ST10_1_DM260_Result_Data_64_bytes_1[23] := HwInputs.ST10_1_DM260_Result_Data_64_bytes_1[23];
	PlcInputs.ST10_1_DM260_Result_Data_64_bytes_1[24] := HwInputs.ST10_1_DM260_Result_Data_64_bytes_1[24];
	PlcInputs.ST10_1_DM260_Result_Data_64_bytes_1[25] := HwInputs.ST10_1_DM260_Result_Data_64_bytes_1[25];
	PlcInputs.ST10_1_DM260_Result_Data_64_bytes_1[26] := HwInputs.ST10_1_DM260_Result_Data_64_bytes_1[26];
	PlcInputs.ST10_1_DM260_Result_Data_64_bytes_1[27] := HwInputs.ST10_1_DM260_Result_Data_64_bytes_1[27];
	PlcInputs.ST10_1_DM260_Result_Data_64_bytes_1[28] := HwInputs.ST10_1_DM260_Result_Data_64_bytes_1[28];
	PlcInputs.ST10_1_DM260_Result_Data_64_bytes_1[29] := HwInputs.ST10_1_DM260_Result_Data_64_bytes_1[29];
	PlcInputs.ST10_1_DM260_Result_Data_64_bytes_1[30] := HwInputs.ST10_1_DM260_Result_Data_64_bytes_1[30];
	PlcInputs.ST10_1_DM260_Result_Data_64_bytes_1[31] := HwInputs.ST10_1_DM260_Result_Data_64_bytes_1[31];
	PlcInputs.ST10_1_DM260_Result_Data_64_bytes_1[32] := HwInputs.ST10_1_DM260_Result_Data_64_bytes_1[32];
	PlcInputs.ST10_1_DM260_Result_Data_64_bytes_1[33] := HwInputs.ST10_1_DM260_Result_Data_64_bytes_1[33];
	PlcInputs.ST10_1_DM260_Result_Data_64_bytes_1[34] := HwInputs.ST10_1_DM260_Result_Data_64_bytes_1[34];
	PlcInputs.ST10_1_DM260_Result_Data_64_bytes_1[35] := HwInputs.ST10_1_DM260_Result_Data_64_bytes_1[35];
	PlcInputs.ST10_1_DM260_Result_Data_64_bytes_1[36] := HwInputs.ST10_1_DM260_Result_Data_64_bytes_1[36];
	PlcInputs.ST10_1_DM260_Result_Data_64_bytes_1[37] := HwInputs.ST10_1_DM260_Result_Data_64_bytes_1[37];
	PlcInputs.ST10_1_DM260_Result_Data_64_bytes_1[38] := HwInputs.ST10_1_DM260_Result_Data_64_bytes_1[38];
	PlcInputs.ST10_1_DM260_Result_Data_64_bytes_1[39] := HwInputs.ST10_1_DM260_Result_Data_64_bytes_1[39];
	PlcInputs.ST10_1_DM260_Result_Data_64_bytes_1[40] := HwInputs.ST10_1_DM260_Result_Data_64_bytes_1[40];
	PlcInputs.ST10_1_DM260_Result_Data_64_bytes_1[41] := HwInputs.ST10_1_DM260_Result_Data_64_bytes_1[41];
	PlcInputs.ST10_1_DM260_Result_Data_64_bytes_1[42] := HwInputs.ST10_1_DM260_Result_Data_64_bytes_1[42];
	PlcInputs.ST10_1_DM260_Result_Data_64_bytes_1[43] := HwInputs.ST10_1_DM260_Result_Data_64_bytes_1[43];
	PlcInputs.ST10_1_DM260_Result_Data_64_bytes_1[44] := HwInputs.ST10_1_DM260_Result_Data_64_bytes_1[44];
	PlcInputs.ST10_1_DM260_Result_Data_64_bytes_1[45] := HwInputs.ST10_1_DM260_Result_Data_64_bytes_1[45];
	PlcInputs.ST10_1_DM260_Result_Data_64_bytes_1[46] := HwInputs.ST10_1_DM260_Result_Data_64_bytes_1[46];
	PlcInputs.ST10_1_DM260_Result_Data_64_bytes_1[47] := HwInputs.ST10_1_DM260_Result_Data_64_bytes_1[47];
	PlcInputs.ST10_1_DM260_Result_Data_64_bytes_1[48] := HwInputs.ST10_1_DM260_Result_Data_64_bytes_1[48];
	PlcInputs.ST10_1_DM260_Result_Data_64_bytes_1[49] := HwInputs.ST10_1_DM260_Result_Data_64_bytes_1[49];
	PlcInputs.ST10_1_DM260_Result_Data_64_bytes_1[50] := HwInputs.ST10_1_DM260_Result_Data_64_bytes_1[50];
	PlcInputs.ST10_1_DM260_Result_Data_64_bytes_1[51] := HwInputs.ST10_1_DM260_Result_Data_64_bytes_1[51];
	PlcInputs.ST10_1_DM260_Result_Data_64_bytes_1[52] := HwInputs.ST10_1_DM260_Result_Data_64_bytes_1[52];
	PlcInputs.ST10_1_DM260_Result_Data_64_bytes_1[53] := HwInputs.ST10_1_DM260_Result_Data_64_bytes_1[53];
	PlcInputs.ST10_1_DM260_Result_Data_64_bytes_1[54] := HwInputs.ST10_1_DM260_Result_Data_64_bytes_1[54];
	PlcInputs.ST10_1_DM260_Result_Data_64_bytes_1[55] := HwInputs.ST10_1_DM260_Result_Data_64_bytes_1[55];
	PlcInputs.ST10_1_DM260_Result_Data_64_bytes_1[56] := HwInputs.ST10_1_DM260_Result_Data_64_bytes_1[56];
	PlcInputs.ST10_1_DM260_Result_Data_64_bytes_1[57] := HwInputs.ST10_1_DM260_Result_Data_64_bytes_1[57];
	PlcInputs.ST10_1_DM260_Result_Data_64_bytes_1[58] := HwInputs.ST10_1_DM260_Result_Data_64_bytes_1[58];
	PlcInputs.ST10_1_DM260_Result_Data_64_bytes_1[59] := HwInputs.ST10_1_DM260_Result_Data_64_bytes_1[59];
	PlcInputs.ST10_1_DM260_Result_Data_64_bytes_1[60] := HwInputs.ST10_1_DM260_Result_Data_64_bytes_1[60];
	PlcInputs.ST10_1_DM260_Result_Data_64_bytes_1[61] := HwInputs.ST10_1_DM260_Result_Data_64_bytes_1[61];
	PlcInputs.ST10_1_DM260_Result_Data_64_bytes_1[62] := HwInputs.ST10_1_DM260_Result_Data_64_bytes_1[62];
	PlcInputs.ST10_1_DM260_Result_Data_64_bytes_1[63] := HwInputs.ST10_1_DM260_Result_Data_64_bytes_1[63];
	PlcInputs.ST10_1_DM260_Result_Data_64_bytes_1[64] := HwInputs.ST10_1_DM260_Result_Data_64_bytes_1[64];
	PlcInputs.ST10_1_DM260_Result_Data_64_bytes_1[65] := HwInputs.ST10_1_DM260_Result_Data_64_bytes_1[65];
	PlcInputs.ST10_1_DM260_Result_Data_64_bytes_1[66] := HwInputs.ST10_1_DM260_Result_Data_64_bytes_1[66];
	PlcInputs.ST10_1_DM260_Result_Data_64_bytes_1[67] := HwInputs.ST10_1_DM260_Result_Data_64_bytes_1[67];
	PlcInputs.ST10_1_DM260_Result_Data_64_bytes_1[68] := HwInputs.ST10_1_DM260_Result_Data_64_bytes_1[68];
	PlcInputs.ST10_1_DM260_Result_Data_64_bytes_1[69] := HwInputs.ST10_1_DM260_Result_Data_64_bytes_1[69];
	PlcInputs.ST10_1_DM260_Result_Data_64_bytes_1[70] := HwInputs.ST10_1_DM260_Result_Data_64_bytes_1[70];
	PlcInputs.ST10_1_DM260_Result_Data_64_bytes_1[71] := HwInputs.ST10_1_DM260_Result_Data_64_bytes_1[71];
	PlcInputs.ST10_1_DM260_Turned_Acquisition_Status_1[0] := HwInputs.ST10_1_DM260_Turned_Acquisition_Status_1[0];
	PlcInputs.ST10_1_DM260_Turned_Acquisition_Status_1[1] := HwInputs.ST10_1_DM260_Turned_Acquisition_Status_1[1];
	PlcInputs.ST10_1_DM260_Turned_Acquisition_Status_1[2] := HwInputs.ST10_1_DM260_Turned_Acquisition_Status_1[2];
	PlcInputs.ST10_1_DM260_Turned_Results_Status_1 := HwInputs.ST10_1_DM260_Turned_Results_Status_1;
	PlcInputs.ST10_1_DM260_Turned_Soft_Event_Control_1 := HwInputs.ST10_1_DM260_Turned_Soft_Event_Control_1;
	PlcInputs.ST10_1_DM260_Turned_Result_Data_64_bytes_1[0] := HwInputs.ST10_1_DM260_Turned_Result_Data_64_bytes_1[0];
	PlcInputs.ST10_1_DM260_Turned_Result_Data_64_bytes_1[1] := HwInputs.ST10_1_DM260_Turned_Result_Data_64_bytes_1[1];
	PlcInputs.ST10_1_DM260_Turned_Result_Data_64_bytes_1[2] := HwInputs.ST10_1_DM260_Turned_Result_Data_64_bytes_1[2];
	PlcInputs.ST10_1_DM260_Turned_Result_Data_64_bytes_1[3] := HwInputs.ST10_1_DM260_Turned_Result_Data_64_bytes_1[3];
	PlcInputs.ST10_1_DM260_Turned_Result_Data_64_bytes_1[4] := HwInputs.ST10_1_DM260_Turned_Result_Data_64_bytes_1[4];
	PlcInputs.ST10_1_DM260_Turned_Result_Data_64_bytes_1[5] := HwInputs.ST10_1_DM260_Turned_Result_Data_64_bytes_1[5];
	PlcInputs.ST10_1_DM260_Turned_Result_Data_64_bytes_1[6] := HwInputs.ST10_1_DM260_Turned_Result_Data_64_bytes_1[6];
	PlcInputs.ST10_1_DM260_Turned_Result_Data_64_bytes_1[7] := HwInputs.ST10_1_DM260_Turned_Result_Data_64_bytes_1[7];
	PlcInputs.ST10_1_DM260_Turned_Result_Data_64_bytes_1[8] := HwInputs.ST10_1_DM260_Turned_Result_Data_64_bytes_1[8];
	PlcInputs.ST10_1_DM260_Turned_Result_Data_64_bytes_1[9] := HwInputs.ST10_1_DM260_Turned_Result_Data_64_bytes_1[9];
	PlcInputs.ST10_1_DM260_Turned_Result_Data_64_bytes_1[10] := HwInputs.ST10_1_DM260_Turned_Result_Data_64_bytes_1[10];
	PlcInputs.ST10_1_DM260_Turned_Result_Data_64_bytes_1[11] := HwInputs.ST10_1_DM260_Turned_Result_Data_64_bytes_1[11];
	PlcInputs.ST10_1_DM260_Turned_Result_Data_64_bytes_1[12] := HwInputs.ST10_1_DM260_Turned_Result_Data_64_bytes_1[12];
	PlcInputs.ST10_1_DM260_Turned_Result_Data_64_bytes_1[13] := HwInputs.ST10_1_DM260_Turned_Result_Data_64_bytes_1[13];
	PlcInputs.ST10_1_DM260_Turned_Result_Data_64_bytes_1[14] := HwInputs.ST10_1_DM260_Turned_Result_Data_64_bytes_1[14];
	PlcInputs.ST10_1_DM260_Turned_Result_Data_64_bytes_1[15] := HwInputs.ST10_1_DM260_Turned_Result_Data_64_bytes_1[15];
	PlcInputs.ST10_1_DM260_Turned_Result_Data_64_bytes_1[16] := HwInputs.ST10_1_DM260_Turned_Result_Data_64_bytes_1[16];
	PlcInputs.ST10_1_DM260_Turned_Result_Data_64_bytes_1[17] := HwInputs.ST10_1_DM260_Turned_Result_Data_64_bytes_1[17];
	PlcInputs.ST10_1_DM260_Turned_Result_Data_64_bytes_1[18] := HwInputs.ST10_1_DM260_Turned_Result_Data_64_bytes_1[18];
	PlcInputs.ST10_1_DM260_Turned_Result_Data_64_bytes_1[19] := HwInputs.ST10_1_DM260_Turned_Result_Data_64_bytes_1[19];
	PlcInputs.ST10_1_DM260_Turned_Result_Data_64_bytes_1[20] := HwInputs.ST10_1_DM260_Turned_Result_Data_64_bytes_1[20];
	PlcInputs.ST10_1_DM260_Turned_Result_Data_64_bytes_1[21] := HwInputs.ST10_1_DM260_Turned_Result_Data_64_bytes_1[21];
	PlcInputs.ST10_1_DM260_Turned_Result_Data_64_bytes_1[22] := HwInputs.ST10_1_DM260_Turned_Result_Data_64_bytes_1[22];
	PlcInputs.ST10_1_DM260_Turned_Result_Data_64_bytes_1[23] := HwInputs.ST10_1_DM260_Turned_Result_Data_64_bytes_1[23];
	PlcInputs.ST10_1_DM260_Turned_Result_Data_64_bytes_1[24] := HwInputs.ST10_1_DM260_Turned_Result_Data_64_bytes_1[24];
	PlcInputs.ST10_1_DM260_Turned_Result_Data_64_bytes_1[25] := HwInputs.ST10_1_DM260_Turned_Result_Data_64_bytes_1[25];
	PlcInputs.ST10_1_DM260_Turned_Result_Data_64_bytes_1[26] := HwInputs.ST10_1_DM260_Turned_Result_Data_64_bytes_1[26];
	PlcInputs.ST10_1_DM260_Turned_Result_Data_64_bytes_1[27] := HwInputs.ST10_1_DM260_Turned_Result_Data_64_bytes_1[27];
	PlcInputs.ST10_1_DM260_Turned_Result_Data_64_bytes_1[28] := HwInputs.ST10_1_DM260_Turned_Result_Data_64_bytes_1[28];
	PlcInputs.ST10_1_DM260_Turned_Result_Data_64_bytes_1[29] := HwInputs.ST10_1_DM260_Turned_Result_Data_64_bytes_1[29];
	PlcInputs.ST10_1_DM260_Turned_Result_Data_64_bytes_1[30] := HwInputs.ST10_1_DM260_Turned_Result_Data_64_bytes_1[30];
	PlcInputs.ST10_1_DM260_Turned_Result_Data_64_bytes_1[31] := HwInputs.ST10_1_DM260_Turned_Result_Data_64_bytes_1[31];
	PlcInputs.ST10_1_DM260_Turned_Result_Data_64_bytes_1[32] := HwInputs.ST10_1_DM260_Turned_Result_Data_64_bytes_1[32];
	PlcInputs.ST10_1_DM260_Turned_Result_Data_64_bytes_1[33] := HwInputs.ST10_1_DM260_Turned_Result_Data_64_bytes_1[33];
	PlcInputs.ST10_1_DM260_Turned_Result_Data_64_bytes_1[34] := HwInputs.ST10_1_DM260_Turned_Result_Data_64_bytes_1[34];
	PlcInputs.ST10_1_DM260_Turned_Result_Data_64_bytes_1[35] := HwInputs.ST10_1_DM260_Turned_Result_Data_64_bytes_1[35];
	PlcInputs.ST10_1_DM260_Turned_Result_Data_64_bytes_1[36] := HwInputs.ST10_1_DM260_Turned_Result_Data_64_bytes_1[36];
	PlcInputs.ST10_1_DM260_Turned_Result_Data_64_bytes_1[37] := HwInputs.ST10_1_DM260_Turned_Result_Data_64_bytes_1[37];
	PlcInputs.ST10_1_DM260_Turned_Result_Data_64_bytes_1[38] := HwInputs.ST10_1_DM260_Turned_Result_Data_64_bytes_1[38];
	PlcInputs.ST10_1_DM260_Turned_Result_Data_64_bytes_1[39] := HwInputs.ST10_1_DM260_Turned_Result_Data_64_bytes_1[39];
	PlcInputs.ST10_1_DM260_Turned_Result_Data_64_bytes_1[40] := HwInputs.ST10_1_DM260_Turned_Result_Data_64_bytes_1[40];
	PlcInputs.ST10_1_DM260_Turned_Result_Data_64_bytes_1[41] := HwInputs.ST10_1_DM260_Turned_Result_Data_64_bytes_1[41];
	PlcInputs.ST10_1_DM260_Turned_Result_Data_64_bytes_1[42] := HwInputs.ST10_1_DM260_Turned_Result_Data_64_bytes_1[42];
	PlcInputs.ST10_1_DM260_Turned_Result_Data_64_bytes_1[43] := HwInputs.ST10_1_DM260_Turned_Result_Data_64_bytes_1[43];
	PlcInputs.ST10_1_DM260_Turned_Result_Data_64_bytes_1[44] := HwInputs.ST10_1_DM260_Turned_Result_Data_64_bytes_1[44];
	PlcInputs.ST10_1_DM260_Turned_Result_Data_64_bytes_1[45] := HwInputs.ST10_1_DM260_Turned_Result_Data_64_bytes_1[45];
	PlcInputs.ST10_1_DM260_Turned_Result_Data_64_bytes_1[46] := HwInputs.ST10_1_DM260_Turned_Result_Data_64_bytes_1[46];
	PlcInputs.ST10_1_DM260_Turned_Result_Data_64_bytes_1[47] := HwInputs.ST10_1_DM260_Turned_Result_Data_64_bytes_1[47];
	PlcInputs.ST10_1_DM260_Turned_Result_Data_64_bytes_1[48] := HwInputs.ST10_1_DM260_Turned_Result_Data_64_bytes_1[48];
	PlcInputs.ST10_1_DM260_Turned_Result_Data_64_bytes_1[49] := HwInputs.ST10_1_DM260_Turned_Result_Data_64_bytes_1[49];
	PlcInputs.ST10_1_DM260_Turned_Result_Data_64_bytes_1[50] := HwInputs.ST10_1_DM260_Turned_Result_Data_64_bytes_1[50];
	PlcInputs.ST10_1_DM260_Turned_Result_Data_64_bytes_1[51] := HwInputs.ST10_1_DM260_Turned_Result_Data_64_bytes_1[51];
	PlcInputs.ST10_1_DM260_Turned_Result_Data_64_bytes_1[52] := HwInputs.ST10_1_DM260_Turned_Result_Data_64_bytes_1[52];
	PlcInputs.ST10_1_DM260_Turned_Result_Data_64_bytes_1[53] := HwInputs.ST10_1_DM260_Turned_Result_Data_64_bytes_1[53];
	PlcInputs.ST10_1_DM260_Turned_Result_Data_64_bytes_1[54] := HwInputs.ST10_1_DM260_Turned_Result_Data_64_bytes_1[54];
	PlcInputs.ST10_1_DM260_Turned_Result_Data_64_bytes_1[55] := HwInputs.ST10_1_DM260_Turned_Result_Data_64_bytes_1[55];
	PlcInputs.ST10_1_DM260_Turned_Result_Data_64_bytes_1[56] := HwInputs.ST10_1_DM260_Turned_Result_Data_64_bytes_1[56];
	PlcInputs.ST10_1_DM260_Turned_Result_Data_64_bytes_1[57] := HwInputs.ST10_1_DM260_Turned_Result_Data_64_bytes_1[57];
	PlcInputs.ST10_1_DM260_Turned_Result_Data_64_bytes_1[58] := HwInputs.ST10_1_DM260_Turned_Result_Data_64_bytes_1[58];
	PlcInputs.ST10_1_DM260_Turned_Result_Data_64_bytes_1[59] := HwInputs.ST10_1_DM260_Turned_Result_Data_64_bytes_1[59];
	PlcInputs.ST10_1_DM260_Turned_Result_Data_64_bytes_1[60] := HwInputs.ST10_1_DM260_Turned_Result_Data_64_bytes_1[60];
	PlcInputs.ST10_1_DM260_Turned_Result_Data_64_bytes_1[61] := HwInputs.ST10_1_DM260_Turned_Result_Data_64_bytes_1[61];
	PlcInputs.ST10_1_DM260_Turned_Result_Data_64_bytes_1[62] := HwInputs.ST10_1_DM260_Turned_Result_Data_64_bytes_1[62];
	PlcInputs.ST10_1_DM260_Turned_Result_Data_64_bytes_1[63] := HwInputs.ST10_1_DM260_Turned_Result_Data_64_bytes_1[63];
	PlcInputs.ST10_1_DM260_Turned_Result_Data_64_bytes_1[64] := HwInputs.ST10_1_DM260_Turned_Result_Data_64_bytes_1[64];
	PlcInputs.ST10_1_DM260_Turned_Result_Data_64_bytes_1[65] := HwInputs.ST10_1_DM260_Turned_Result_Data_64_bytes_1[65];
	PlcInputs.ST10_1_DM260_Turned_Result_Data_64_bytes_1[66] := HwInputs.ST10_1_DM260_Turned_Result_Data_64_bytes_1[66];
	PlcInputs.ST10_1_DM260_Turned_Result_Data_64_bytes_1[67] := HwInputs.ST10_1_DM260_Turned_Result_Data_64_bytes_1[67];
	PlcInputs.ST10_1_DM260_Turned_Result_Data_64_bytes_1[68] := HwInputs.ST10_1_DM260_Turned_Result_Data_64_bytes_1[68];
	PlcInputs.ST10_1_DM260_Turned_Result_Data_64_bytes_1[69] := HwInputs.ST10_1_DM260_Turned_Result_Data_64_bytes_1[69];
	PlcInputs.ST10_1_DM260_Turned_Result_Data_64_bytes_1[70] := HwInputs.ST10_1_DM260_Turned_Result_Data_64_bytes_1[70];
	PlcInputs.ST10_1_DM260_Turned_Result_Data_64_bytes_1[71] := HwInputs.ST10_1_DM260_Turned_Result_Data_64_bytes_1[71];
END_FUNCTION

(* ---- CopyOutputs.st ---- *)
FUNCTION CopyOutputs
	VAR_EXTERNAL
		HwOutputs : HwOutputs;
		PlcOutputs : PlcOutputs;
	END_VAR
	HwOutputs.ST10_ET200SP_CM_AS_i_Master_ST_1[0] := PlcOutputs.ST10_ET200SP_CM_AS_i_Master_ST_1[0];
	HwOutputs.ST10_ET200SP_CM_AS_i_Master_ST_1[1] := PlcOutputs.ST10_ET200SP_CM_AS_i_Master_ST_1[1];
	HwOutputs.ST10_ET200SP_CM_AS_i_Master_ST_1[2] := PlcOutputs.ST10_ET200SP_CM_AS_i_Master_ST_1[2];
	HwOutputs.ST10_ET200SP_CM_AS_i_Master_ST_1[3] := PlcOutputs.ST10_ET200SP_CM_AS_i_Master_ST_1[3];
	HwOutputs.ST10_ET200SP_CM_AS_i_Master_ST_1[4] := PlcOutputs.ST10_ET200SP_CM_AS_i_Master_ST_1[4];
	HwOutputs.ST10_ET200SP_CM_AS_i_Master_ST_1[5] := PlcOutputs.ST10_ET200SP_CM_AS_i_Master_ST_1[5];
	HwOutputs.ST10_ET200SP_CM_AS_i_Master_ST_1[6] := PlcOutputs.ST10_ET200SP_CM_AS_i_Master_ST_1[6];
	HwOutputs.ST10_ET200SP_CM_AS_i_Master_ST_1[7] := PlcOutputs.ST10_ET200SP_CM_AS_i_Master_ST_1[7];
	HwOutputs.ST10_ET200SP_CM_AS_i_Master_ST_1[8] := PlcOutputs.ST10_ET200SP_CM_AS_i_Master_ST_1[8];
	HwOutputs.ST10_ET200SP_CM_AS_i_Master_ST_1[9] := PlcOutputs.ST10_ET200SP_CM_AS_i_Master_ST_1[9];
	HwOutputs.ST10_ET200SP_CM_AS_i_Master_ST_1[10] := PlcOutputs.ST10_ET200SP_CM_AS_i_Master_ST_1[10];
	HwOutputs.ST10_ET200SP_CM_AS_i_Master_ST_1[11] := PlcOutputs.ST10_ET200SP_CM_AS_i_Master_ST_1[11];
	HwOutputs.ST10_ET200SP_CM_AS_i_Master_ST_1[12] := PlcOutputs.ST10_ET200SP_CM_AS_i_Master_ST_1[12];
	HwOutputs.ST10_ET200SP_CM_AS_i_Master_ST_1[13] := PlcOutputs.ST10_ET200SP_CM_AS_i_Master_ST_1[13];
	HwOutputs.ST10_ET200SP_CM_AS_i_Master_ST_1[14] := PlcOutputs.ST10_ET200SP_CM_AS_i_Master_ST_1[14];
	HwOutputs.ST10_ET200SP_CM_AS_i_Master_ST_1[15] := PlcOutputs.ST10_ET200SP_CM_AS_i_Master_ST_1[15];
	HwOutputs.ST10_ET200SP_CM_AS_i_Master_ST_1[16] := PlcOutputs.ST10_ET200SP_CM_AS_i_Master_ST_1[16];
	HwOutputs.ST10_ET200SP_CM_AS_i_Master_ST_1[17] := PlcOutputs.ST10_ET200SP_CM_AS_i_Master_ST_1[17];
	HwOutputs.ST10_ET200SP_CM_AS_i_Master_ST_1[18] := PlcOutputs.ST10_ET200SP_CM_AS_i_Master_ST_1[18];
	HwOutputs.ST10_ET200SP_CM_AS_i_Master_ST_1[19] := PlcOutputs.ST10_ET200SP_CM_AS_i_Master_ST_1[19];
	HwOutputs.ST10_ET200SP_CM_AS_i_Master_ST_1[20] := PlcOutputs.ST10_ET200SP_CM_AS_i_Master_ST_1[20];
	HwOutputs.ST10_ET200SP_CM_AS_i_Master_ST_1[21] := PlcOutputs.ST10_ET200SP_CM_AS_i_Master_ST_1[21];
	HwOutputs.ST10_ET200SP_CM_AS_i_Master_ST_1[22] := PlcOutputs.ST10_ET200SP_CM_AS_i_Master_ST_1[22];
	HwOutputs.ST10_ET200SP_CM_AS_i_Master_ST_1[23] := PlcOutputs.ST10_ET200SP_CM_AS_i_Master_ST_1[23];
	HwOutputs.ST10_ET200SP_CM_AS_i_Master_ST_1[24] := PlcOutputs.ST10_ET200SP_CM_AS_i_Master_ST_1[24];
	HwOutputs.ST10_ET200SP_CM_AS_i_Master_ST_1[25] := PlcOutputs.ST10_ET200SP_CM_AS_i_Master_ST_1[25];
	HwOutputs.ST10_ET200SP_CM_AS_i_Master_ST_1[26] := PlcOutputs.ST10_ET200SP_CM_AS_i_Master_ST_1[26];
	HwOutputs.ST10_ET200SP_CM_AS_i_Master_ST_1[27] := PlcOutputs.ST10_ET200SP_CM_AS_i_Master_ST_1[27];
	HwOutputs.ST10_ET200SP_CM_AS_i_Master_ST_1[28] := PlcOutputs.ST10_ET200SP_CM_AS_i_Master_ST_1[28];
	HwOutputs.ST10_ET200SP_CM_AS_i_Master_ST_1[29] := PlcOutputs.ST10_ET200SP_CM_AS_i_Master_ST_1[29];
	HwOutputs.ST10_ET200SP_CM_AS_i_Master_ST_1[30] := PlcOutputs.ST10_ET200SP_CM_AS_i_Master_ST_1[30];
	HwOutputs.ST10_ET200SP_CM_AS_i_Master_ST_1[31] := PlcOutputs.ST10_ET200SP_CM_AS_i_Master_ST_1[31];
	HwOutputs.ST10_ET200SP_CM_AS_i_Master_ST_1[32] := PlcOutputs.ST10_ET200SP_CM_AS_i_Master_ST_1[32];
	HwOutputs.ST10_ET200SP_CM_AS_i_Master_ST_1[33] := PlcOutputs.ST10_ET200SP_CM_AS_i_Master_ST_1[33];
	HwOutputs.ST10_ET200SP_CM_AS_i_Master_ST_1[34] := PlcOutputs.ST10_ET200SP_CM_AS_i_Master_ST_1[34];
	HwOutputs.ST10_ET200SP_CM_AS_i_Master_ST_1[35] := PlcOutputs.ST10_ET200SP_CM_AS_i_Master_ST_1[35];
	HwOutputs.ST10_ET200SP_CM_AS_i_Master_ST_1[36] := PlcOutputs.ST10_ET200SP_CM_AS_i_Master_ST_1[36];
	HwOutputs.ST10_ET200SP_CM_AS_i_Master_ST_1[37] := PlcOutputs.ST10_ET200SP_CM_AS_i_Master_ST_1[37];
	HwOutputs.ST10_ET200SP_CM_AS_i_Master_ST_1[38] := PlcOutputs.ST10_ET200SP_CM_AS_i_Master_ST_1[38];
	HwOutputs.ST10_ET200SP_CM_AS_i_Master_ST_1[39] := PlcOutputs.ST10_ET200SP_CM_AS_i_Master_ST_1[39];
	HwOutputs.ST10_ET200SP_CM_AS_i_Master_ST_1[40] := PlcOutputs.ST10_ET200SP_CM_AS_i_Master_ST_1[40];
	HwOutputs.ST10_ET200SP_CM_AS_i_Master_ST_1[41] := PlcOutputs.ST10_ET200SP_CM_AS_i_Master_ST_1[41];
	HwOutputs.ST10_ET200SP_CM_AS_i_Master_ST_1[42] := PlcOutputs.ST10_ET200SP_CM_AS_i_Master_ST_1[42];
	HwOutputs.ST10_ET200SP_CM_AS_i_Master_ST_1[43] := PlcOutputs.ST10_ET200SP_CM_AS_i_Master_ST_1[43];
	HwOutputs.ST10_ET200SP_CM_AS_i_Master_ST_1[44] := PlcOutputs.ST10_ET200SP_CM_AS_i_Master_ST_1[44];
	HwOutputs.ST10_ET200SP_CM_AS_i_Master_ST_1[45] := PlcOutputs.ST10_ET200SP_CM_AS_i_Master_ST_1[45];
	HwOutputs.ST10_ET200SP_CM_AS_i_Master_ST_1[46] := PlcOutputs.ST10_ET200SP_CM_AS_i_Master_ST_1[46];
	HwOutputs.ST10_ET200SP_CM_AS_i_Master_ST_1[47] := PlcOutputs.ST10_ET200SP_CM_AS_i_Master_ST_1[47];
	HwOutputs.ST10_ET200SP_CM_AS_i_Master_ST_1[48] := PlcOutputs.ST10_ET200SP_CM_AS_i_Master_ST_1[48];
	HwOutputs.ST10_ET200SP_CM_AS_i_Master_ST_1[49] := PlcOutputs.ST10_ET200SP_CM_AS_i_Master_ST_1[49];
	HwOutputs.ST10_ET200SP_CM_AS_i_Master_ST_1[50] := PlcOutputs.ST10_ET200SP_CM_AS_i_Master_ST_1[50];
	HwOutputs.ST10_ET200SP_CM_AS_i_Master_ST_1[51] := PlcOutputs.ST10_ET200SP_CM_AS_i_Master_ST_1[51];
	HwOutputs.ST10_ET200SP_CM_AS_i_Master_ST_1[52] := PlcOutputs.ST10_ET200SP_CM_AS_i_Master_ST_1[52];
	HwOutputs.ST10_ET200SP_CM_AS_i_Master_ST_1[53] := PlcOutputs.ST10_ET200SP_CM_AS_i_Master_ST_1[53];
	HwOutputs.ST10_ET200SP_CM_AS_i_Master_ST_1[54] := PlcOutputs.ST10_ET200SP_CM_AS_i_Master_ST_1[54];
	HwOutputs.ST10_ET200SP_CM_AS_i_Master_ST_1[55] := PlcOutputs.ST10_ET200SP_CM_AS_i_Master_ST_1[55];
	HwOutputs.ST10_ET200SP_CM_AS_i_Master_ST_1[56] := PlcOutputs.ST10_ET200SP_CM_AS_i_Master_ST_1[56];
	HwOutputs.ST10_ET200SP_CM_AS_i_Master_ST_1[57] := PlcOutputs.ST10_ET200SP_CM_AS_i_Master_ST_1[57];
	HwOutputs.ST10_ET200SP_CM_AS_i_Master_ST_1[58] := PlcOutputs.ST10_ET200SP_CM_AS_i_Master_ST_1[58];
	HwOutputs.ST10_ET200SP_CM_AS_i_Master_ST_1[59] := PlcOutputs.ST10_ET200SP_CM_AS_i_Master_ST_1[59];
	HwOutputs.ST10_ET200SP_CM_AS_i_Master_ST_1[60] := PlcOutputs.ST10_ET200SP_CM_AS_i_Master_ST_1[60];
	HwOutputs.ST10_ET200SP_CM_AS_i_Master_ST_1[61] := PlcOutputs.ST10_ET200SP_CM_AS_i_Master_ST_1[61];
	HwOutputs.ST10_ET200SP_CM_AS_i_Master_ST_1[62] := PlcOutputs.ST10_ET200SP_CM_AS_i_Master_ST_1[62];
	HwOutputs.ST10_ET200SP_CM_AS_i_Master_ST_1[63] := PlcOutputs.ST10_ET200SP_CM_AS_i_Master_ST_1[63];
	HwOutputs.ST10_ET200SP_DQ_8x24VDC_0_5A_ST_1 := PlcOutputs.ST10_ET200SP_DQ_8x24VDC_0_5A_ST_1;
	HwOutputs.ST10_ET200SP_DQ_8x24VDC_0_5A_ST_2 := PlcOutputs.ST10_ET200SP_DQ_8x24VDC_0_5A_ST_2;
	HwOutputs.ST10_ET200SP_DQ_8x24VDC_0_5A_ST_3 := PlcOutputs.ST10_ET200SP_DQ_8x24VDC_0_5A_ST_3;
	HwOutputs.ST10_ET200SP_DQ_8x24VDC_0_5A_ST_4 := PlcOutputs.ST10_ET200SP_DQ_8x24VDC_0_5A_ST_4;
	HwOutputs.ST10_ET200SP_CM_4xIO_Link_1[0] := PlcOutputs.ST10_ET200SP_CM_4xIO_Link_1[0];
	HwOutputs.ST10_ET200SP_CM_4xIO_Link_1[1] := PlcOutputs.ST10_ET200SP_CM_4xIO_Link_1[1];
	HwOutputs.ST10_ET200SP_CM_4xIO_Link_1[2] := PlcOutputs.ST10_ET200SP_CM_4xIO_Link_1[2];
	HwOutputs.ST10_ET200SP_CM_4xIO_Link_1[3] := PlcOutputs.ST10_ET200SP_CM_4xIO_Link_1[3];
	HwOutputs.ST10_ET200SP_CM_4xIO_Link_1[4] := PlcOutputs.ST10_ET200SP_CM_4xIO_Link_1[4];
	HwOutputs.ST10_ET200SP_CM_4xIO_Link_1[5] := PlcOutputs.ST10_ET200SP_CM_4xIO_Link_1[5];
	HwOutputs.ST10_ET200SP_CM_4xIO_Link_1[6] := PlcOutputs.ST10_ET200SP_CM_4xIO_Link_1[6];
	HwOutputs.ST10_ET200SP_CM_4xIO_Link_1[7] := PlcOutputs.ST10_ET200SP_CM_4xIO_Link_1[7];
	HwOutputs.ST10_ET200SP_CM_4xIO_Link_1[8] := PlcOutputs.ST10_ET200SP_CM_4xIO_Link_1[8];
	HwOutputs.ST10_ET200SP_CM_4xIO_Link_1[9] := PlcOutputs.ST10_ET200SP_CM_4xIO_Link_1[9];
	HwOutputs.ST10_ET200SP_CM_4xIO_Link_1[10] := PlcOutputs.ST10_ET200SP_CM_4xIO_Link_1[10];
	HwOutputs.ST10_ET200SP_CM_4xIO_Link_1[11] := PlcOutputs.ST10_ET200SP_CM_4xIO_Link_1[11];
	HwOutputs.ST10_ET200SP_CM_4xIO_Link_1[12] := PlcOutputs.ST10_ET200SP_CM_4xIO_Link_1[12];
	HwOutputs.ST10_ET200SP_CM_4xIO_Link_1[13] := PlcOutputs.ST10_ET200SP_CM_4xIO_Link_1[13];
	HwOutputs.ST10_ET200SP_CM_4xIO_Link_1[14] := PlcOutputs.ST10_ET200SP_CM_4xIO_Link_1[14];
	HwOutputs.ST10_ET200SP_CM_4xIO_Link_1[15] := PlcOutputs.ST10_ET200SP_CM_4xIO_Link_1[15];
	HwOutputs.ST10_ET200SP_CM_4xIO_Link_1[16] := PlcOutputs.ST10_ET200SP_CM_4xIO_Link_1[16];
	HwOutputs.ST10_ET200SP_CM_4xIO_Link_1[17] := PlcOutputs.ST10_ET200SP_CM_4xIO_Link_1[17];
	HwOutputs.ST10_ET200SP_CM_4xIO_Link_1[18] := PlcOutputs.ST10_ET200SP_CM_4xIO_Link_1[18];
	HwOutputs.ST10_ET200SP_CM_4xIO_Link_1[19] := PlcOutputs.ST10_ET200SP_CM_4xIO_Link_1[19];
	HwOutputs.ST10_ET200SP_CM_4xIO_Link_1[20] := PlcOutputs.ST10_ET200SP_CM_4xIO_Link_1[20];
	HwOutputs.ST10_ET200SP_CM_4xIO_Link_1[21] := PlcOutputs.ST10_ET200SP_CM_4xIO_Link_1[21];
	HwOutputs.ST10_ET200SP_CM_4xIO_Link_1[22] := PlcOutputs.ST10_ET200SP_CM_4xIO_Link_1[22];
	HwOutputs.ST10_ET200SP_CM_4xIO_Link_1[23] := PlcOutputs.ST10_ET200SP_CM_4xIO_Link_1[23];
	HwOutputs.ST10_ET200SP_CM_4xIO_Link_1[24] := PlcOutputs.ST10_ET200SP_CM_4xIO_Link_1[24];
	HwOutputs.ST10_ET200SP_CM_4xIO_Link_1[25] := PlcOutputs.ST10_ET200SP_CM_4xIO_Link_1[25];
	HwOutputs.ST10_ET200SP_CM_4xIO_Link_1[26] := PlcOutputs.ST10_ET200SP_CM_4xIO_Link_1[26];
	HwOutputs.ST10_ET200SP_CM_4xIO_Link_1[27] := PlcOutputs.ST10_ET200SP_CM_4xIO_Link_1[27];
	HwOutputs.ST10_ET200SP_CM_4xIO_Link_1[28] := PlcOutputs.ST10_ET200SP_CM_4xIO_Link_1[28];
	HwOutputs.ST10_ET200SP_CM_4xIO_Link_1[29] := PlcOutputs.ST10_ET200SP_CM_4xIO_Link_1[29];
	HwOutputs.ST10_ET200SP_CM_4xIO_Link_1[30] := PlcOutputs.ST10_ET200SP_CM_4xIO_Link_1[30];
	HwOutputs.ST10_ET200SP_CM_4xIO_Link_1[31] := PlcOutputs.ST10_ET200SP_CM_4xIO_Link_1[31];
	HwOutputs.ST10_ET200SP_2_21FM1 := PlcOutputs.ST10_ET200SP_2_21FM1;
	HwOutputs.ST10_ET200SP_2_21FM2 := PlcOutputs.ST10_ET200SP_2_21FM2;
	HwOutputs.ST10_ET200SP_2_21FM3 := PlcOutputs.ST10_ET200SP_2_21FM3;
	HwOutputs.ST10_ET200SP_2_21FM4 := PlcOutputs.ST10_ET200SP_2_21FM4;
	HwOutputs.ST10_ET200SP_2_21FM5 := PlcOutputs.ST10_ET200SP_2_21FM5;
	HwOutputs.ST10_ET200SP_2_21FM6 := PlcOutputs.ST10_ET200SP_2_21FM6;
	HwOutputs.ST10_ET200SP_2_21FM7 := PlcOutputs.ST10_ET200SP_2_21FM7;
	HwOutputs.ST10_ET200SP_2_21FM8 := PlcOutputs.ST10_ET200SP_2_21FM8;
	HwOutputs.ST10_ET200SP_2_21FM9 := PlcOutputs.ST10_ET200SP_2_21FM9;
	HwOutputs.ST10_ET200SP_2_21FM10 := PlcOutputs.ST10_ET200SP_2_21FM10;
	HwOutputs.ST10_ET200SP_2_21FM11 := PlcOutputs.ST10_ET200SP_2_21FM11;
	HwOutputs.ST10_ET200SP_2_21FM12 := PlcOutputs.ST10_ET200SP_2_21FM12;
	HwOutputs.ST10_ET200SP_2_22FM1 := PlcOutputs.ST10_ET200SP_2_22FM1;
	HwOutputs.ST10_ET200SP_2_22FM2 := PlcOutputs.ST10_ET200SP_2_22FM2;
	HwOutputs.ST10_ET200SP_2_22FM3 := PlcOutputs.ST10_ET200SP_2_22FM3;
	HwOutputs.ST10_ET200SP_2_22FM4 := PlcOutputs.ST10_ET200SP_2_22FM4;
	HwOutputs.ST10_ET200SP_2_22FM5 := PlcOutputs.ST10_ET200SP_2_22FM5;
	HwOutputs.ST10_ET200SP_2_22FM6 := PlcOutputs.ST10_ET200SP_2_22FM6;
	HwOutputs.ST10_ET200SP_2_22FM7 := PlcOutputs.ST10_ET200SP_2_22FM7;
	HwOutputs.ST10_ET200SP_2_22FM8 := PlcOutputs.ST10_ET200SP_2_22FM8;
	HwOutputs.ST10_ET200SP_2_22FM9 := PlcOutputs.ST10_ET200SP_2_22FM9;
	HwOutputs.ST10_ET200SP_2_22FM10 := PlcOutputs.ST10_ET200SP_2_22FM10;
	HwOutputs.ST10_ET200SP_2_22FM11 := PlcOutputs.ST10_ET200SP_2_22FM11;
	HwOutputs.ST10_ET200SP_2_22FM12 := PlcOutputs.ST10_ET200SP_2_22FM12;
	HwOutputs.ST10_ET200SP_2_22FM13 := PlcOutputs.ST10_ET200SP_2_22FM13;
	HwOutputs.ST10_CPX_MPA1S_VMPA1_FB_EMS_8_8DO_1 := PlcOutputs.ST10_CPX_MPA1S_VMPA1_FB_EMS_8_8DO_1;
	HwOutputs.ST10_CPX_MPA2G_VMPA2_FB_EMG_4_4DO_1 := PlcOutputs.ST10_CPX_MPA2G_VMPA2_FB_EMG_4_4DO_1;
	HwOutputs.ST10_1_DM260_Acquisition_Control_1 := PlcOutputs.ST10_1_DM260_Acquisition_Control_1;
	HwOutputs.ST10_1_DM260_Results_Control_1 := PlcOutputs.ST10_1_DM260_Results_Control_1;
	HwOutputs.ST10_1_DM260_Soft_Event_Control_1 := PlcOutputs.ST10_1_DM260_Soft_Event_Control_1;
	HwOutputs.ST10_1_DM260_User_Data_64_bytes_1[0] := PlcOutputs.ST10_1_DM260_User_Data_64_bytes_1[0];
	HwOutputs.ST10_1_DM260_User_Data_64_bytes_1[1] := PlcOutputs.ST10_1_DM260_User_Data_64_bytes_1[1];
	HwOutputs.ST10_1_DM260_User_Data_64_bytes_1[2] := PlcOutputs.ST10_1_DM260_User_Data_64_bytes_1[2];
	HwOutputs.ST10_1_DM260_User_Data_64_bytes_1[3] := PlcOutputs.ST10_1_DM260_User_Data_64_bytes_1[3];
	HwOutputs.ST10_1_DM260_User_Data_64_bytes_1[4] := PlcOutputs.ST10_1_DM260_User_Data_64_bytes_1[4];
	HwOutputs.ST10_1_DM260_User_Data_64_bytes_1[5] := PlcOutputs.ST10_1_DM260_User_Data_64_bytes_1[5];
	HwOutputs.ST10_1_DM260_User_Data_64_bytes_1[6] := PlcOutputs.ST10_1_DM260_User_Data_64_bytes_1[6];
	HwOutputs.ST10_1_DM260_User_Data_64_bytes_1[7] := PlcOutputs.ST10_1_DM260_User_Data_64_bytes_1[7];
	HwOutputs.ST10_1_DM260_User_Data_64_bytes_1[8] := PlcOutputs.ST10_1_DM260_User_Data_64_bytes_1[8];
	HwOutputs.ST10_1_DM260_User_Data_64_bytes_1[9] := PlcOutputs.ST10_1_DM260_User_Data_64_bytes_1[9];
	HwOutputs.ST10_1_DM260_User_Data_64_bytes_1[10] := PlcOutputs.ST10_1_DM260_User_Data_64_bytes_1[10];
	HwOutputs.ST10_1_DM260_User_Data_64_bytes_1[11] := PlcOutputs.ST10_1_DM260_User_Data_64_bytes_1[11];
	HwOutputs.ST10_1_DM260_User_Data_64_bytes_1[12] := PlcOutputs.ST10_1_DM260_User_Data_64_bytes_1[12];
	HwOutputs.ST10_1_DM260_User_Data_64_bytes_1[13] := PlcOutputs.ST10_1_DM260_User_Data_64_bytes_1[13];
	HwOutputs.ST10_1_DM260_User_Data_64_bytes_1[14] := PlcOutputs.ST10_1_DM260_User_Data_64_bytes_1[14];
	HwOutputs.ST10_1_DM260_User_Data_64_bytes_1[15] := PlcOutputs.ST10_1_DM260_User_Data_64_bytes_1[15];
	HwOutputs.ST10_1_DM260_User_Data_64_bytes_1[16] := PlcOutputs.ST10_1_DM260_User_Data_64_bytes_1[16];
	HwOutputs.ST10_1_DM260_User_Data_64_bytes_1[17] := PlcOutputs.ST10_1_DM260_User_Data_64_bytes_1[17];
	HwOutputs.ST10_1_DM260_User_Data_64_bytes_1[18] := PlcOutputs.ST10_1_DM260_User_Data_64_bytes_1[18];
	HwOutputs.ST10_1_DM260_User_Data_64_bytes_1[19] := PlcOutputs.ST10_1_DM260_User_Data_64_bytes_1[19];
	HwOutputs.ST10_1_DM260_User_Data_64_bytes_1[20] := PlcOutputs.ST10_1_DM260_User_Data_64_bytes_1[20];
	HwOutputs.ST10_1_DM260_User_Data_64_bytes_1[21] := PlcOutputs.ST10_1_DM260_User_Data_64_bytes_1[21];
	HwOutputs.ST10_1_DM260_User_Data_64_bytes_1[22] := PlcOutputs.ST10_1_DM260_User_Data_64_bytes_1[22];
	HwOutputs.ST10_1_DM260_User_Data_64_bytes_1[23] := PlcOutputs.ST10_1_DM260_User_Data_64_bytes_1[23];
	HwOutputs.ST10_1_DM260_User_Data_64_bytes_1[24] := PlcOutputs.ST10_1_DM260_User_Data_64_bytes_1[24];
	HwOutputs.ST10_1_DM260_User_Data_64_bytes_1[25] := PlcOutputs.ST10_1_DM260_User_Data_64_bytes_1[25];
	HwOutputs.ST10_1_DM260_User_Data_64_bytes_1[26] := PlcOutputs.ST10_1_DM260_User_Data_64_bytes_1[26];
	HwOutputs.ST10_1_DM260_User_Data_64_bytes_1[27] := PlcOutputs.ST10_1_DM260_User_Data_64_bytes_1[27];
	HwOutputs.ST10_1_DM260_User_Data_64_bytes_1[28] := PlcOutputs.ST10_1_DM260_User_Data_64_bytes_1[28];
	HwOutputs.ST10_1_DM260_User_Data_64_bytes_1[29] := PlcOutputs.ST10_1_DM260_User_Data_64_bytes_1[29];
	HwOutputs.ST10_1_DM260_User_Data_64_bytes_1[30] := PlcOutputs.ST10_1_DM260_User_Data_64_bytes_1[30];
	HwOutputs.ST10_1_DM260_User_Data_64_bytes_1[31] := PlcOutputs.ST10_1_DM260_User_Data_64_bytes_1[31];
	HwOutputs.ST10_1_DM260_User_Data_64_bytes_1[32] := PlcOutputs.ST10_1_DM260_User_Data_64_bytes_1[32];
	HwOutputs.ST10_1_DM260_User_Data_64_bytes_1[33] := PlcOutputs.ST10_1_DM260_User_Data_64_bytes_1[33];
	HwOutputs.ST10_1_DM260_User_Data_64_bytes_1[34] := PlcOutputs.ST10_1_DM260_User_Data_64_bytes_1[34];
	HwOutputs.ST10_1_DM260_User_Data_64_bytes_1[35] := PlcOutputs.ST10_1_DM260_User_Data_64_bytes_1[35];
	HwOutputs.ST10_1_DM260_User_Data_64_bytes_1[36] := PlcOutputs.ST10_1_DM260_User_Data_64_bytes_1[36];
	HwOutputs.ST10_1_DM260_User_Data_64_bytes_1[37] := PlcOutputs.ST10_1_DM260_User_Data_64_bytes_1[37];
	HwOutputs.ST10_1_DM260_User_Data_64_bytes_1[38] := PlcOutputs.ST10_1_DM260_User_Data_64_bytes_1[38];
	HwOutputs.ST10_1_DM260_User_Data_64_bytes_1[39] := PlcOutputs.ST10_1_DM260_User_Data_64_bytes_1[39];
	HwOutputs.ST10_1_DM260_User_Data_64_bytes_1[40] := PlcOutputs.ST10_1_DM260_User_Data_64_bytes_1[40];
	HwOutputs.ST10_1_DM260_User_Data_64_bytes_1[41] := PlcOutputs.ST10_1_DM260_User_Data_64_bytes_1[41];
	HwOutputs.ST10_1_DM260_User_Data_64_bytes_1[42] := PlcOutputs.ST10_1_DM260_User_Data_64_bytes_1[42];
	HwOutputs.ST10_1_DM260_User_Data_64_bytes_1[43] := PlcOutputs.ST10_1_DM260_User_Data_64_bytes_1[43];
	HwOutputs.ST10_1_DM260_User_Data_64_bytes_1[44] := PlcOutputs.ST10_1_DM260_User_Data_64_bytes_1[44];
	HwOutputs.ST10_1_DM260_User_Data_64_bytes_1[45] := PlcOutputs.ST10_1_DM260_User_Data_64_bytes_1[45];
	HwOutputs.ST10_1_DM260_User_Data_64_bytes_1[46] := PlcOutputs.ST10_1_DM260_User_Data_64_bytes_1[46];
	HwOutputs.ST10_1_DM260_User_Data_64_bytes_1[47] := PlcOutputs.ST10_1_DM260_User_Data_64_bytes_1[47];
	HwOutputs.ST10_1_DM260_User_Data_64_bytes_1[48] := PlcOutputs.ST10_1_DM260_User_Data_64_bytes_1[48];
	HwOutputs.ST10_1_DM260_User_Data_64_bytes_1[49] := PlcOutputs.ST10_1_DM260_User_Data_64_bytes_1[49];
	HwOutputs.ST10_1_DM260_User_Data_64_bytes_1[50] := PlcOutputs.ST10_1_DM260_User_Data_64_bytes_1[50];
	HwOutputs.ST10_1_DM260_User_Data_64_bytes_1[51] := PlcOutputs.ST10_1_DM260_User_Data_64_bytes_1[51];
	HwOutputs.ST10_1_DM260_User_Data_64_bytes_1[52] := PlcOutputs.ST10_1_DM260_User_Data_64_bytes_1[52];
	HwOutputs.ST10_1_DM260_User_Data_64_bytes_1[53] := PlcOutputs.ST10_1_DM260_User_Data_64_bytes_1[53];
	HwOutputs.ST10_1_DM260_User_Data_64_bytes_1[54] := PlcOutputs.ST10_1_DM260_User_Data_64_bytes_1[54];
	HwOutputs.ST10_1_DM260_User_Data_64_bytes_1[55] := PlcOutputs.ST10_1_DM260_User_Data_64_bytes_1[55];
	HwOutputs.ST10_1_DM260_User_Data_64_bytes_1[56] := PlcOutputs.ST10_1_DM260_User_Data_64_bytes_1[56];
	HwOutputs.ST10_1_DM260_User_Data_64_bytes_1[57] := PlcOutputs.ST10_1_DM260_User_Data_64_bytes_1[57];
	HwOutputs.ST10_1_DM260_User_Data_64_bytes_1[58] := PlcOutputs.ST10_1_DM260_User_Data_64_bytes_1[58];
	HwOutputs.ST10_1_DM260_User_Data_64_bytes_1[59] := PlcOutputs.ST10_1_DM260_User_Data_64_bytes_1[59];
	HwOutputs.ST10_1_DM260_User_Data_64_bytes_1[60] := PlcOutputs.ST10_1_DM260_User_Data_64_bytes_1[60];
	HwOutputs.ST10_1_DM260_User_Data_64_bytes_1[61] := PlcOutputs.ST10_1_DM260_User_Data_64_bytes_1[61];
	HwOutputs.ST10_1_DM260_User_Data_64_bytes_1[62] := PlcOutputs.ST10_1_DM260_User_Data_64_bytes_1[62];
	HwOutputs.ST10_1_DM260_User_Data_64_bytes_1[63] := PlcOutputs.ST10_1_DM260_User_Data_64_bytes_1[63];
	HwOutputs.ST10_1_DM260_User_Data_64_bytes_1[64] := PlcOutputs.ST10_1_DM260_User_Data_64_bytes_1[64];
	HwOutputs.ST10_1_DM260_User_Data_64_bytes_1[65] := PlcOutputs.ST10_1_DM260_User_Data_64_bytes_1[65];
	HwOutputs.ST10_1_DM260_User_Data_64_bytes_1[66] := PlcOutputs.ST10_1_DM260_User_Data_64_bytes_1[66];
	HwOutputs.ST10_1_DM260_User_Data_64_bytes_1[67] := PlcOutputs.ST10_1_DM260_User_Data_64_bytes_1[67];
	HwOutputs.ST10_1_DM260_Turned_Acquisition_Control_1 := PlcOutputs.ST10_1_DM260_Turned_Acquisition_Control_1;
	HwOutputs.ST10_1_DM260_Turned_Results_Control_1 := PlcOutputs.ST10_1_DM260_Turned_Results_Control_1;
	HwOutputs.ST10_1_DM260_Turned_Soft_Event_Control_1 := PlcOutputs.ST10_1_DM260_Turned_Soft_Event_Control_1;
	HwOutputs.ST10_1_DM260_Turned_User_Data_64_bytes_1[0] := PlcOutputs.ST10_1_DM260_Turned_User_Data_64_bytes_1[0];
	HwOutputs.ST10_1_DM260_Turned_User_Data_64_bytes_1[1] := PlcOutputs.ST10_1_DM260_Turned_User_Data_64_bytes_1[1];
	HwOutputs.ST10_1_DM260_Turned_User_Data_64_bytes_1[2] := PlcOutputs.ST10_1_DM260_Turned_User_Data_64_bytes_1[2];
	HwOutputs.ST10_1_DM260_Turned_User_Data_64_bytes_1[3] := PlcOutputs.ST10_1_DM260_Turned_User_Data_64_bytes_1[3];
	HwOutputs.ST10_1_DM260_Turned_User_Data_64_bytes_1[4] := PlcOutputs.ST10_1_DM260_Turned_User_Data_64_bytes_1[4];
	HwOutputs.ST10_1_DM260_Turned_User_Data_64_bytes_1[5] := PlcOutputs.ST10_1_DM260_Turned_User_Data_64_bytes_1[5];
	HwOutputs.ST10_1_DM260_Turned_User_Data_64_bytes_1[6] := PlcOutputs.ST10_1_DM260_Turned_User_Data_64_bytes_1[6];
	HwOutputs.ST10_1_DM260_Turned_User_Data_64_bytes_1[7] := PlcOutputs.ST10_1_DM260_Turned_User_Data_64_bytes_1[7];
	HwOutputs.ST10_1_DM260_Turned_User_Data_64_bytes_1[8] := PlcOutputs.ST10_1_DM260_Turned_User_Data_64_bytes_1[8];
	HwOutputs.ST10_1_DM260_Turned_User_Data_64_bytes_1[9] := PlcOutputs.ST10_1_DM260_Turned_User_Data_64_bytes_1[9];
	HwOutputs.ST10_1_DM260_Turned_User_Data_64_bytes_1[10] := PlcOutputs.ST10_1_DM260_Turned_User_Data_64_bytes_1[10];
	HwOutputs.ST10_1_DM260_Turned_User_Data_64_bytes_1[11] := PlcOutputs.ST10_1_DM260_Turned_User_Data_64_bytes_1[11];
	HwOutputs.ST10_1_DM260_Turned_User_Data_64_bytes_1[12] := PlcOutputs.ST10_1_DM260_Turned_User_Data_64_bytes_1[12];
	HwOutputs.ST10_1_DM260_Turned_User_Data_64_bytes_1[13] := PlcOutputs.ST10_1_DM260_Turned_User_Data_64_bytes_1[13];
	HwOutputs.ST10_1_DM260_Turned_User_Data_64_bytes_1[14] := PlcOutputs.ST10_1_DM260_Turned_User_Data_64_bytes_1[14];
	HwOutputs.ST10_1_DM260_Turned_User_Data_64_bytes_1[15] := PlcOutputs.ST10_1_DM260_Turned_User_Data_64_bytes_1[15];
	HwOutputs.ST10_1_DM260_Turned_User_Data_64_bytes_1[16] := PlcOutputs.ST10_1_DM260_Turned_User_Data_64_bytes_1[16];
	HwOutputs.ST10_1_DM260_Turned_User_Data_64_bytes_1[17] := PlcOutputs.ST10_1_DM260_Turned_User_Data_64_bytes_1[17];
	HwOutputs.ST10_1_DM260_Turned_User_Data_64_bytes_1[18] := PlcOutputs.ST10_1_DM260_Turned_User_Data_64_bytes_1[18];
	HwOutputs.ST10_1_DM260_Turned_User_Data_64_bytes_1[19] := PlcOutputs.ST10_1_DM260_Turned_User_Data_64_bytes_1[19];
	HwOutputs.ST10_1_DM260_Turned_User_Data_64_bytes_1[20] := PlcOutputs.ST10_1_DM260_Turned_User_Data_64_bytes_1[20];
	HwOutputs.ST10_1_DM260_Turned_User_Data_64_bytes_1[21] := PlcOutputs.ST10_1_DM260_Turned_User_Data_64_bytes_1[21];
	HwOutputs.ST10_1_DM260_Turned_User_Data_64_bytes_1[22] := PlcOutputs.ST10_1_DM260_Turned_User_Data_64_bytes_1[22];
	HwOutputs.ST10_1_DM260_Turned_User_Data_64_bytes_1[23] := PlcOutputs.ST10_1_DM260_Turned_User_Data_64_bytes_1[23];
	HwOutputs.ST10_1_DM260_Turned_User_Data_64_bytes_1[24] := PlcOutputs.ST10_1_DM260_Turned_User_Data_64_bytes_1[24];
	HwOutputs.ST10_1_DM260_Turned_User_Data_64_bytes_1[25] := PlcOutputs.ST10_1_DM260_Turned_User_Data_64_bytes_1[25];
	HwOutputs.ST10_1_DM260_Turned_User_Data_64_bytes_1[26] := PlcOutputs.ST10_1_DM260_Turned_User_Data_64_bytes_1[26];
	HwOutputs.ST10_1_DM260_Turned_User_Data_64_bytes_1[27] := PlcOutputs.ST10_1_DM260_Turned_User_Data_64_bytes_1[27];
	HwOutputs.ST10_1_DM260_Turned_User_Data_64_bytes_1[28] := PlcOutputs.ST10_1_DM260_Turned_User_Data_64_bytes_1[28];
	HwOutputs.ST10_1_DM260_Turned_User_Data_64_bytes_1[29] := PlcOutputs.ST10_1_DM260_Turned_User_Data_64_bytes_1[29];
	HwOutputs.ST10_1_DM260_Turned_User_Data_64_bytes_1[30] := PlcOutputs.ST10_1_DM260_Turned_User_Data_64_bytes_1[30];
	HwOutputs.ST10_1_DM260_Turned_User_Data_64_bytes_1[31] := PlcOutputs.ST10_1_DM260_Turned_User_Data_64_bytes_1[31];
	HwOutputs.ST10_1_DM260_Turned_User_Data_64_bytes_1[32] := PlcOutputs.ST10_1_DM260_Turned_User_Data_64_bytes_1[32];
	HwOutputs.ST10_1_DM260_Turned_User_Data_64_bytes_1[33] := PlcOutputs.ST10_1_DM260_Turned_User_Data_64_bytes_1[33];
	HwOutputs.ST10_1_DM260_Turned_User_Data_64_bytes_1[34] := PlcOutputs.ST10_1_DM260_Turned_User_Data_64_bytes_1[34];
	HwOutputs.ST10_1_DM260_Turned_User_Data_64_bytes_1[35] := PlcOutputs.ST10_1_DM260_Turned_User_Data_64_bytes_1[35];
	HwOutputs.ST10_1_DM260_Turned_User_Data_64_bytes_1[36] := PlcOutputs.ST10_1_DM260_Turned_User_Data_64_bytes_1[36];
	HwOutputs.ST10_1_DM260_Turned_User_Data_64_bytes_1[37] := PlcOutputs.ST10_1_DM260_Turned_User_Data_64_bytes_1[37];
	HwOutputs.ST10_1_DM260_Turned_User_Data_64_bytes_1[38] := PlcOutputs.ST10_1_DM260_Turned_User_Data_64_bytes_1[38];
	HwOutputs.ST10_1_DM260_Turned_User_Data_64_bytes_1[39] := PlcOutputs.ST10_1_DM260_Turned_User_Data_64_bytes_1[39];
	HwOutputs.ST10_1_DM260_Turned_User_Data_64_bytes_1[40] := PlcOutputs.ST10_1_DM260_Turned_User_Data_64_bytes_1[40];
	HwOutputs.ST10_1_DM260_Turned_User_Data_64_bytes_1[41] := PlcOutputs.ST10_1_DM260_Turned_User_Data_64_bytes_1[41];
	HwOutputs.ST10_1_DM260_Turned_User_Data_64_bytes_1[42] := PlcOutputs.ST10_1_DM260_Turned_User_Data_64_bytes_1[42];
	HwOutputs.ST10_1_DM260_Turned_User_Data_64_bytes_1[43] := PlcOutputs.ST10_1_DM260_Turned_User_Data_64_bytes_1[43];
	HwOutputs.ST10_1_DM260_Turned_User_Data_64_bytes_1[44] := PlcOutputs.ST10_1_DM260_Turned_User_Data_64_bytes_1[44];
	HwOutputs.ST10_1_DM260_Turned_User_Data_64_bytes_1[45] := PlcOutputs.ST10_1_DM260_Turned_User_Data_64_bytes_1[45];
	HwOutputs.ST10_1_DM260_Turned_User_Data_64_bytes_1[46] := PlcOutputs.ST10_1_DM260_Turned_User_Data_64_bytes_1[46];
	HwOutputs.ST10_1_DM260_Turned_User_Data_64_bytes_1[47] := PlcOutputs.ST10_1_DM260_Turned_User_Data_64_bytes_1[47];
	HwOutputs.ST10_1_DM260_Turned_User_Data_64_bytes_1[48] := PlcOutputs.ST10_1_DM260_Turned_User_Data_64_bytes_1[48];
	HwOutputs.ST10_1_DM260_Turned_User_Data_64_bytes_1[49] := PlcOutputs.ST10_1_DM260_Turned_User_Data_64_bytes_1[49];
	HwOutputs.ST10_1_DM260_Turned_User_Data_64_bytes_1[50] := PlcOutputs.ST10_1_DM260_Turned_User_Data_64_bytes_1[50];
	HwOutputs.ST10_1_DM260_Turned_User_Data_64_bytes_1[51] := PlcOutputs.ST10_1_DM260_Turned_User_Data_64_bytes_1[51];
	HwOutputs.ST10_1_DM260_Turned_User_Data_64_bytes_1[52] := PlcOutputs.ST10_1_DM260_Turned_User_Data_64_bytes_1[52];
	HwOutputs.ST10_1_DM260_Turned_User_Data_64_bytes_1[53] := PlcOutputs.ST10_1_DM260_Turned_User_Data_64_bytes_1[53];
	HwOutputs.ST10_1_DM260_Turned_User_Data_64_bytes_1[54] := PlcOutputs.ST10_1_DM260_Turned_User_Data_64_bytes_1[54];
	HwOutputs.ST10_1_DM260_Turned_User_Data_64_bytes_1[55] := PlcOutputs.ST10_1_DM260_Turned_User_Data_64_bytes_1[55];
	HwOutputs.ST10_1_DM260_Turned_User_Data_64_bytes_1[56] := PlcOutputs.ST10_1_DM260_Turned_User_Data_64_bytes_1[56];
	HwOutputs.ST10_1_DM260_Turned_User_Data_64_bytes_1[57] := PlcOutputs.ST10_1_DM260_Turned_User_Data_64_bytes_1[57];
	HwOutputs.ST10_1_DM260_Turned_User_Data_64_bytes_1[58] := PlcOutputs.ST10_1_DM260_Turned_User_Data_64_bytes_1[58];
	HwOutputs.ST10_1_DM260_Turned_User_Data_64_bytes_1[59] := PlcOutputs.ST10_1_DM260_Turned_User_Data_64_bytes_1[59];
	HwOutputs.ST10_1_DM260_Turned_User_Data_64_bytes_1[60] := PlcOutputs.ST10_1_DM260_Turned_User_Data_64_bytes_1[60];
	HwOutputs.ST10_1_DM260_Turned_User_Data_64_bytes_1[61] := PlcOutputs.ST10_1_DM260_Turned_User_Data_64_bytes_1[61];
	HwOutputs.ST10_1_DM260_Turned_User_Data_64_bytes_1[62] := PlcOutputs.ST10_1_DM260_Turned_User_Data_64_bytes_1[62];
	HwOutputs.ST10_1_DM260_Turned_User_Data_64_bytes_1[63] := PlcOutputs.ST10_1_DM260_Turned_User_Data_64_bytes_1[63];
	HwOutputs.ST10_1_DM260_Turned_User_Data_64_bytes_1[64] := PlcOutputs.ST10_1_DM260_Turned_User_Data_64_bytes_1[64];
	HwOutputs.ST10_1_DM260_Turned_User_Data_64_bytes_1[65] := PlcOutputs.ST10_1_DM260_Turned_User_Data_64_bytes_1[65];
	HwOutputs.ST10_1_DM260_Turned_User_Data_64_bytes_1[66] := PlcOutputs.ST10_1_DM260_Turned_User_Data_64_bytes_1[66];
	HwOutputs.ST10_1_DM260_Turned_User_Data_64_bytes_1[67] := PlcOutputs.ST10_1_DM260_Turned_User_Data_64_bytes_1[67];
END_FUNCTION
